LIN {X 0,Y 467.549,Z 320.867,A -85,B 0,C 180,E1 -7525.167,E2 -7525.167} C_VEL
LIN {X 0,Y 467.574,Z 320.867,A -85,B 0,C 180,E1 -7528.26,E2 -7528.26} C_VEL
LIN {X 0,Y 467.538,Z 320.867,A -85,B 0,C 180,E1 -7531.248,E2 -7531.248} C_VEL
LIN {X 0,Y 467.578,Z 320.87,A -85,B 0,C 180,E1 -7534.401,E2 -7534.401} C_VEL
LIN {X 0,Y 467.552,Z 320.866,A -85,B 0,C 180,E1 -7536.995,E2 -7536.995} C_VEL
LIN {X 0,Y 467.613,Z 320.859,A -85,B 0,C 180,E1 -7539.777,E2 -7539.777} C_VEL
LIN {X 0,Y 467.566,Z 320.868,A -85,B 0,C 180,E1 -7542.505,E2 -7542.505} C_VEL
LIN {X 0,Y 467.593,Z 320.86,A -85,B 0,C 180,E1 -7545.196,E2 -7545.196} C_VEL
LIN {X 0,Y 467.658,Z 320.855,A -85,B 0,C 180,E1 -7547.855,E2 -7547.855} C_VEL
LIN {X 0,Y 467.669,Z 320.851,A -85,B 0,C 180,E1 -7551.357,E2 -7551.357} C_VEL
LIN {X 0,Y 467.719,Z 320.851,A -85,B 0,C 180,E1 -7553.963,E2 -7553.963} C_VEL
LIN {X 0,Y 467.852,Z 320.829,A -85,B 0,C 180,E1 -7557.417,E2 -7557.417} C_VEL
LIN {X 0,Y 467.881,Z 320.832,A -85,B 0,C 180,E1 -7560,E2 -7560} C_VEL
LIN {X 0,Y 467.85,Z 320.829,A -85,B 0,C 180,E1 -7562.583,E2 -7562.583} C_VEL
LIN {X 0,Y 467.723,Z 320.85,A -85,B 0,C 180,E1 -7566.038,E2 -7566.038} C_VEL
LIN {X 0,Y 467.683,Z 320.849,A -85,B 0,C 180,E1 -7568.643,E2 -7568.643} C_VEL
LIN {X 0,Y 467.658,Z 320.853,A -85,B 0,C 180,E1 -7572.358,E2 -7572.358} C_VEL
LIN {X 0,Y 467.653,Z 320.858,A -85,B 0,C 180,E1 -7575.885,E2 -7575.885} C_VEL
LIN {X 0,Y 467.627,Z 320.859,A -85,B 0,C 180,E1 -7579.308,E2 -7579.308} C_VEL
LIN {X 0,Y 467.538,Z 320.869,A -85,B 0,C 180,E1 -7582.074,E2 -7582.074} C_VEL
LIN {X 0,Y 467.589,Z 320.861,A -85,B 0,C 180,E1 -7584.888,E2 -7584.888} C_VEL
LIN {X 0,Y 467.624,Z 320.861,A -85,B 0,C 180,E1 -7587.769,E2 -7587.769} C_VEL
LIN {X 0,Y 467.572,Z 320.865,A -85,B 0,C 180,E1 -7591.045,E2 -7591.045} C_VEL
LIN {X 0,Y 467.591,Z 320.86,A -85,B 0,C 180,E1 -7594.242,E2 -7594.242} C_VEL
LIN {X 0,Y 467.546,Z 320.871,A -85,B 0,C 180,E1 -7597.185,E2 -7597.185} C_VEL
LIN {X 0,Y 467.581,Z 320.861,A -85,B 0,C 180,E1 -7600.264,E2 -7600.264} C_VEL
LIN {X 0,Y 467.591,Z 320.861,A -85,B 0,C 180,E1 -7602.567,E2 -7602.567} C_VEL
LIN {X 0,Y 467.574,Z 320.868,A -85,B 0,C 180,E1 -7605.053,E2 -7605.053} C_VEL
LIN {X 0,Y 467.593,Z 320.865,A -85,B 0,C 180,E1 -7607.44,E2 -7607.44} C_VEL
LIN {X 0,Y 467.586,Z 320.865,A -85,B 0,C 180,E1 -7610.855,E2 -7610.855} C_VEL
LIN {X 0,Y 467.564,Z 320.864,A -85,B 0,C 180,E1 -7614.261,E2 -7614.261} C_VEL
LIN {X 0,Y 467.586,Z 320.867,A -85,B 0,C 180,E1 -7617.321,E2 -7617.321} C_VEL
LIN {X 0,Y 467.573,Z 320.872,A -85,B 0,C 180,E1 -7620.667,E2 -7620.667} C_VEL
LIN {X 0,Y 467.642,Z 320.956,A -85,B 0,C 180,E1 -7621.714,E2 -7621.714} C_VEL
LIN {X 0,Y 470.915,Z 336.083,A -85,B 0,C 180,E1 -7624.354,E2 -7624.354} C_VEL
LIN {X 0,Y 470.576,Z 345.926,A -85,B 0,C 180,E1 -7625.915,E2 -7625.915} C_VEL
LIN {X 0,Y 469.657,Z 365.378,A -85,B 0,C 180,E1 -7628.952,E2 -7628.952} C_VEL
LIN {X 0,Y 469.514,Z 368.376,A -85,B 0,C 180,E1 -7629.416,E2 -7629.416} C_VEL
LIN {X 0,Y 473.317,Z 391.092,A -85,B 0,C 180,E1 -7629.937,E2 -7629.937} C_VEL
LIN {X 0,Y 472.11,Z 506.208,A -85,B 0,C 180,E1 -7631.726,E2 -7631.726} C_VEL
LIN {X 0,Y 471.675,Z 521.021,A -85,B 0,C 180,E1 -7632.13,E2 -7632.13} C_VEL
LIN {X 0,Y 471.143,Z 534.853,A -85,B 0,C 180,E1 -7632.686,E2 -7632.686} C_VEL
LIN {X 0,Y 470.514,Z 548.55,A -85,B 0,C 180,E1 -7633.425,E2 -7633.425} C_VEL
LIN {X 0,Y 469.856,Z 560.834,A -85,B 0,C 180,E1 -7634.269,E2 -7634.269} C_VEL
LIN {X 0,Y 469.176,Z 572.39,A -85,B 0,C 180,E1 -7635.246,E2 -7635.246} C_VEL
LIN {X 0,Y 468.566,Z 582.999,A -85,B 0,C 180,E1 -7636.335,E2 -7636.335} C_VEL
LIN {X 0,Y 468.11,Z 592.848,A -85,B 0,C 180,E1 -7637.552,E2 -7637.552} C_VEL
LIN {X 0,Y 467.575,Z 602.232,A -85,B 0,C 180,E1 -7638.951,E2 -7638.951} C_VEL
LIN {X 0,Y 467.175,Z 610.555,A -85,B 0,C 180,E1 -7640.474,E2 -7640.474} C_VEL
LIN {X 0,Y 466.931,Z 616.367,A -85,B 0,C 180,E1 -7641.778,E2 -7641.778} C_VEL
LIN {X 0,Y 466.801,Z 621.141,A -85,B 0,C 180,E1 -7643.081,E2 -7643.081} C_VEL
LIN {X 0,Y 466.729,Z 626.083,A -85,B 0,C 180,E1 -7644.816,E2 -7644.816} C_VEL
LIN {X 0,Y 466.681,Z 629.517,A -85,B 0,C 180,E1 -7646.546,E2 -7646.546} C_VEL
LIN {X 0,Y 466.629,Z 631.547,A -85,B 0,C 180,E1 -7648.273,E2 -7648.273} C_VEL
LIN {X 0,Y 466.597,Z 632.219,A -85,B 0,C 180,E1 -7649.999,E2 -7649.999} C_VEL
LIN {X 0,Y 466.629,Z 631.545,A -85,B 0,C 180,E1 -7651.725,E2 -7651.725} C_VEL
LIN {X 0,Y 466.681,Z 629.513,A -85,B 0,C 180,E1 -7653.453,E2 -7653.453} C_VEL
LIN {X 0,Y 466.73,Z 626.075,A -85,B 0,C 180,E1 -7655.183,E2 -7655.183} C_VEL
LIN {X 0,Y 466.821,Z 621.129,A -85,B 0,C 180,E1 -7656.917,E2 -7656.917} C_VEL
LIN {X 0,Y 466.997,Z 614.534,A -85,B 0,C 180,E1 -7658.655,E2 -7658.655} C_VEL
LIN {X 0,Y 467.29,Z 607.208,A -85,B 0,C 180,E1 -7660.178,E2 -7660.178} C_VEL
LIN {X 0,Y 467.782,Z 598.156,A -85,B 0,C 180,E1 -7661.701,E2 -7661.701} C_VEL
LIN {X 0,Y 468.297,Z 588.667,A -85,B 0,C 180,E1 -7663.009,E2 -7663.009} C_VEL
LIN {X 0,Y 468.85,Z 578.175,A -85,B 0,C 180,E1 -7664.208,E2 -7664.208} C_VEL
LIN {X 0,Y 469.579,Z 566.617,A -85,B 0,C 180,E1 -7665.294,E2 -7665.294} C_VEL
LIN {X 0,Y 470.318,Z 553.814,A -85,B 0,C 180,E1 -7666.27,E2 -7666.27} C_VEL
LIN {X 0,Y 470.942,Z 541.697,A -85,B 0,C 180,E1 -7667.009,E2 -7667.009} C_VEL
LIN {X 0,Y 471.5,Z 527.504,A -85,B 0,C 180,E1 -7667.679,E2 -7667.679} C_VEL
LIN {X 0,Y 472.075,Z 513.044,A -85,B 0,C 180,E1 -7668.161,E2 -7668.161} C_VEL
LIN {X 0,Y 472.405,Z 498.853,A -85,B 0,C 180,E1 -7668.457,E2 -7668.457} C_VEL
LIN {X 0,Y 473.422,Z 390.059,A -85,B 0,C 180,E1 -7670.149,E2 -7670.149} C_VEL
LIN {X 0,Y 469.586,Z 368.039,A -85,B 0,C 180,E1 -7670.692,E2 -7670.692} C_VEL
LIN {X 0,Y 470.566,Z 349.91,A -85,B 0,C 180,E1 -7673.547,E2 -7673.547} C_VEL
LIN {X 0,Y 471.099,Z 336.963,A -85,B 0,C 180,E1 -7675.634,E2 -7675.634} C_VEL
LIN {X 0,Y 468.366,Z 324.027,A -85,B 0,C 180,E1 -7677.962,E2 -7677.962} C_VEL
LIN {X 0,Y 467.606,Z 320.864,A -85,B 0,C 180,E1 -7678.562,E2 -7678.562} C_VEL
LIN {X 0,Y 467.581,Z 320.864,A -85,B 0,C 180,E1 -7681.739,E2 -7681.739} C_VEL
LIN {X 0,Y 467.566,Z 320.871,A -85,B 0,C 180,E1 -7684.831,E2 -7684.831} C_VEL
LIN {X 0,Y 467.566,Z 320.866,A -85,B 0,C 180,E1 -7688.043,E2 -7688.043} C_VEL
LIN {X 0,Y 467.59,Z 320.865,A -85,B 0,C 180,E1 -7690.262,E2 -7690.262} C_VEL
LIN {X 0,Y 467.582,Z 320.862,A -85,B 0,C 180,E1 -7692.566,E2 -7692.566} C_VEL
LIN {X 0,Y 467.566,Z 320.862,A -85,B 0,C 180,E1 -7695.052,E2 -7695.052} C_VEL
LIN {X 0,Y 467.584,Z 320.863,A -85,B 0,C 180,E1 -7697.439,E2 -7697.439} C_VEL
LIN {X 0,Y 467.577,Z 320.861,A -85,B 0,C 180,E1 -7700.854,E2 -7700.854} C_VEL
LIN {X 0,Y 467.557,Z 320.869,A -85,B 0,C 180,E1 -7704.26,E2 -7704.26} C_VEL
LIN {X 0,Y 467.575,Z 320.861,A -85,B 0,C 180,E1 -7707.32,E2 -7707.32} C_VEL
LIN {X 0,Y 467.572,Z 320.867,A -85,B 0,C 180,E1 -7710.665,E2 -7710.665} C_VEL
LIN {X 0,Y 467.619,Z 320.855,A -85,B 0,C 180,E1 -7713.2,E2 -7713.2} C_VEL
LIN {X 0,Y 467.584,Z 320.863,A -85,B 0,C 180,E1 -7716.468,E2 -7716.468} C_VEL
LIN {X 0,Y 467.615,Z 320.862,A -85,B 0,C 180,E1 -7719.777,E2 -7719.777} C_VEL
LIN {X 0,Y 467.601,Z 320.863,A -85,B 0,C 180,E1 -7722.506,E2 -7722.506} C_VEL
LIN {X 0,Y 467.597,Z 320.856,A -85,B 0,C 180,E1 -7725.196,E2 -7725.196} C_VEL
LIN {X 0,Y 467.647,Z 320.86,A -85,B 0,C 180,E1 -7727.854,E2 -7727.854} C_VEL
LIN {X 0,Y 467.67,Z 320.853,A -85,B 0,C 180,E1 -7731.357,E2 -7731.357} C_VEL
LIN {X 0,Y 467.723,Z 320.849,A -85,B 0,C 180,E1 -7733.962,E2 -7733.962} C_VEL
LIN {X 0,Y 467.811,Z 320.834,A -85,B 0,C 180,E1 -7737.417,E2 -7737.417} C_VEL
LIN {X 0,Y 467.839,Z 320.832,A -85,B 0,C 180,E1 -7740,E2 -7740} C_VEL
LIN {X 0,Y 467.837,Z 320.83,A -85,B 0,C 180,E1 -7742.583,E2 -7742.583} C_VEL
LIN {X 0,Y 467.683,Z 320.852,A -85,B 0,C 180,E1 -7746.038,E2 -7746.038} C_VEL
LIN {X 0,Y 467.624,Z 320.855,A -85,B 0,C 180,E1 -7748.644,E2 -7748.644} C_VEL
LIN {X 0,Y 467.645,Z 320.852,A -85,B 0,C 180,E1 -7752.145,E2 -7752.145} C_VEL
LIN {X 0,Y 467.612,Z 320.858,A -85,B 0,C 180,E1 -7755.873,E2 -7755.873} C_VEL
LIN {X 0,Y 467.608,Z 320.863,A -85,B 0,C 180,E1 -7759.308,E2 -7759.308} C_VEL
LIN {X 0,Y 467.52,Z 320.868,A -85,B 0,C 180,E1 -7762.074,E2 -7762.074} C_VEL
LIN {X 0,Y 467.558,Z 320.87,A -85,B 0,C 180,E1 -7764.89,E2 -7764.89} C_VEL
LIN {X 0,Y 467.552,Z 320.863,A -85,B 0,C 180,E1 -7767.773,E2 -7767.773} C_VEL
LIN {X 0,Y 467.555,Z 320.876,A -85,B 0,C 180,E1 -7771.044,E2 -7771.044} C_VEL
LIN {X 0,Y 467.567,Z 320.867,A -85,B 0,C 180,E1 -7774.24,E2 -7774.24} C_VEL
LIN {X 0,Y 467.538,Z 320.872,A -85,B 0,C 180,E1 -7777.187,E2 -7777.187} C_VEL
LIN {X 0,Y 467.566,Z 320.865,A -85,B 0,C 180,E1 -7780.265,E2 -7780.265} C_VEL
LIN {X 0,Y 467.578,Z 320.865,A -85,B 0,C 180,E1 -7782.567,E2 -7782.567} C_VEL
LIN {X 0,Y 467.557,Z 320.871,A -85,B 0,C 180,E1 -7785.053,E2 -7785.053} C_VEL
LIN {X 0,Y 467.623,Z 321.03,A -85,B 0,C 180,E1 -7788.184,E2 -7788.184} C_VEL
LIN {X 0,Y 469.868,Z 332.052,A -85,B 0,C 180,E1 -7790.531,E2 -7790.531} C_VEL
LIN {X 0,Y 469.882,Z 336.532,A -85,B 0,C 180,E1 -7791.386,E2 -7791.386} C_VEL
LIN {X 0,Y 473.693,Z 353.213,A -85,B 0,C 180,E1 -7791.844,E2 -7791.844} C_VEL
LIN {X 0,Y 472.479,Z 472.361,A -85,B 0,C 180,E1 -7793.721,E2 -7793.721} C_VEL
LIN {X 0,Y 472.092,Z 486.72,A -85,B 0,C 180,E1 -7794.115,E2 -7794.115} C_VEL
LIN {X 0,Y 471.664,Z 500.331,A -85,B 0,C 180,E1 -7794.666,E2 -7794.666} C_VEL
LIN {X 0,Y 471.228,Z 510.399,A -85,B 0,C 180,E1 -7795.189,E2 -7795.189} C_VEL
LIN {X 0,Y 470.402,Z 515.734,A -85,B 0,C 180,E1 -7795.48,E2 -7795.48} C_VEL
LIN {X 0,Y 467.231,Z 524.272,A -85,B 0,C 180,E1 -7795.959,E2 -7795.959} C_VEL
LIN {X 0,Y 463.936,Z 532.468,A -85,B 0,C 180,E1 -7796.514,E2 -7796.514} C_VEL
LIN {X 0,Y 462.926,Z 537.249,A -85,B 0,C 180,E1 -7796.923,E2 -7796.923} C_VEL
LIN {X 0,Y 462.295,Z 547.807,A -85,B 0,C 180,E1 -7798.021,E2 -7798.021} C_VEL
LIN {X 0,Y 461.603,Z 558.262,A -85,B 0,C 180,E1 -7799.334,E2 -7799.334} C_VEL
LIN {X 0,Y 460.96,Z 567.82,A -85,B 0,C 180,E1 -7800.799,E2 -7800.799} C_VEL
LIN {X 0,Y 460.489,Z 575.654,A -85,B 0,C 180,E1 -7802.275,E2 -7802.275} C_VEL
LIN {X 0,Y 460.121,Z 581.847,A -85,B 0,C 180,E1 -7803.709,E2 -7803.709} C_VEL
LIN {X 0,Y 459.901,Z 586.868,A -85,B 0,C 180,E1 -7805.151,E2 -7805.151} C_VEL
LIN {X 0,Y 459.725,Z 590.787,A -85,B 0,C 180,E1 -7806.581,E2 -7806.581} C_VEL
LIN {X 0,Y 459.556,Z 594.49,A -85,B 0,C 180,E1 -7808.468,E2 -7808.468} C_VEL
LIN {X 0,Y 459.491,Z 596.599,A -85,B 0,C 180,E1 -7810.338,E2 -7810.338} C_VEL
LIN {X 0,Y 459.481,Z 597.172,A -85,B 0,C 180,E1 -7812.188,E2 -7812.188} C_VEL
LIN {X 0,Y 459.454,Z 596.31,A -85,B 0,C 180,E1 -7814.019,E2 -7814.019} C_VEL
LIN {X 0,Y 459.544,Z 594.028,A -85,B 0,C 180,E1 -7815.837,E2 -7815.837} C_VEL
LIN {X 0,Y 459.75,Z 590.297,A -85,B 0,C 180,E1 -7817.643,E2 -7817.643} C_VEL
LIN {X 0,Y 459.96,Z 585.044,A -85,B 0,C 180,E1 -7819.436,E2 -7819.436} C_VEL
LIN {X 0,Y 460.2,Z 579.947,A -85,B 0,C 180,E1 -7820.774,E2 -7820.774} C_VEL
LIN {X 0,Y 460.54,Z 573.802,A -85,B 0,C 180,E1 -7822.107,E2 -7822.107} C_VEL
LIN {X 0,Y 461.059,Z 565.093,A -85,B 0,C 180,E1 -7823.656,E2 -7823.656} C_VEL
LIN {X 0,Y 461.579,Z 556.016,A -85,B 0,C 180,E1 -7824.978,E2 -7824.978} C_VEL
LIN {X 0,Y 462.27,Z 545.023,A -85,B 0,C 180,E1 -7826.296,E2 -7826.296} C_VEL
LIN {X 0,Y 462.964,Z 533.821,A -85,B 0,C 180,E1 -7827.391,E2 -7827.391} C_VEL
LIN {X 0,Y 463.685,Z 521.54,A -85,B 0,C 180,E1 -7828.367,E2 -7828.367} C_VEL
LIN {X 0,Y 464.295,Z 509.57,A -85,B 0,C 180,E1 -7829.133,E2 -7829.133} C_VEL
LIN {X 0,Y 464.848,Z 496.574,A -85,B 0,C 180,E1 -7829.784,E2 -7829.784} C_VEL
LIN {X 0,Y 465.285,Z 482.579,A -85,B 0,C 180,E1 -7830.298,E2 -7830.298} C_VEL
LIN {X 0,Y 465.603,Z 467.783,A -85,B 0,C 180,E1 -7830.649,E2 -7830.649} C_VEL
LIN {X 0,Y 466.765,Z 354.137,A -85,B 0,C 180,E1 -7832.433,E2 -7832.433} C_VEL
LIN {X 0,Y 462.828,Z 336.193,A -85,B 0,C 180,E1 -7832.917,E2 -7832.917} C_VEL
LIN {X 0,Y 462.659,Z 332.235,A -85,B 0,C 180,E1 -7833.702,E2 -7833.702} C_VEL
LIN {X 0,Y 460.676,Z 321.729,A -85,B 0,C 180,E1 -7835.911,E2 -7835.911} C_VEL
LIN {X 0,Y 460.615,Z 321.735,A -85,B 0,C 180,E1 -7838.777,E2 -7838.777} C_VEL
LIN {X 0,Y 460.595,Z 321.732,A -85,B 0,C 180,E1 -7842.436,E2 -7842.436} C_VEL
LIN {X 0,Y 460.599,Z 321.732,A -85,B 0,C 180,E1 -7845.998,E2 -7845.998} C_VEL
LIN {X 0,Y 460.566,Z 321.738,A -85,B 0,C 180,E1 -7849.616,E2 -7849.616} C_VEL
LIN {X 0,Y 460.505,Z 321.744,A -85,B 0,C 180,E1 -7852.43,E2 -7852.43} C_VEL
LIN {X 0,Y 460.531,Z 321.74,A -85,B 0,C 180,E1 -7855.793,E2 -7855.793} C_VEL
LIN {X 0,Y 460.513,Z 321.747,A -85,B 0,C 180,E1 -7859.233,E2 -7859.233} C_VEL
LIN {X 0,Y 460.497,Z 321.745,A -85,B 0,C 180,E1 -7862.288,E2 -7862.288} C_VEL
LIN {X 0,Y 460.497,Z 321.746,A -85,B 0,C 180,E1 -7865.447,E2 -7865.447} C_VEL
LIN {X 0,Y 460.488,Z 321.753,A -85,B 0,C 180,E1 -7868.89,E2 -7868.89} C_VEL
LIN {X 0,Y 460.5,Z 321.744,A -85,B 0,C 180,E1 -7871.599,E2 -7871.599} C_VEL
LIN {X 0,Y 460.509,Z 321.748,A -85,B 0,C 180,E1 -7874.59,E2 -7874.59} C_VEL
LIN {X 0,Y 460.471,Z 321.747,A -85,B 0,C 180,E1 -7877.813,E2 -7877.813} C_VEL
LIN {X 0,Y 460.475,Z 321.749,A -85,B 0,C 180,E1 -7880.132,E2 -7880.132} C_VEL
LIN {X 0,Y 460.457,Z 321.749,A -85,B 0,C 180,E1 -7883.469,E2 -7883.469} C_VEL
LIN {X 0,Y 460.516,Z 321.748,A -85,B 0,C 180,E1 -7886.675,E2 -7886.675} C_VEL
LIN {X 0,Y 460.496,Z 321.745,A -85,B 0,C 180,E1 -7889.759,E2 -7889.759} C_VEL
LIN {X 0,Y 460.49,Z 321.749,A -85,B 0,C 180,E1 -7892.751,E2 -7892.751} C_VEL
LIN {X 0,Y 460.516,Z 321.742,A -85,B 0,C 180,E1 -7895.667,E2 -7895.667} C_VEL
LIN {X 0,Y 460.52,Z 321.746,A -85,B 0,C 180,E1 -7898.58,E2 -7898.58} C_VEL
LIN {X 0,Y 460.584,Z 321.733,A -85,B 0,C 180,E1 -7901.311,E2 -7901.311} C_VEL
LIN {X 0,Y 460.55,Z 321.738,A -85,B 0,C 180,E1 -7904.965,E2 -7904.965} C_VEL
LIN {X 0,Y 460.611,Z 321.733,A -85,B 0,C 180,E1 -7908.56,E2 -7908.56} C_VEL
LIN {X 0,Y 460.62,Z 321.729,A -85,B 0,C 180,E1 -7911.224,E2 -7911.224} C_VEL
LIN {X 0,Y 460.683,Z 321.726,A -85,B 0,C 180,E1 -7913.87,E2 -7913.87} C_VEL
LIN {X 0,Y 460.793,Z 321.708,A -85,B 0,C 180,E1 -7917.378,E2 -7917.378} C_VEL
LIN {X 0,Y 460.85,Z 321.708,A -85,B 0,C 180,E1 -7920,E2 -7920} C_VEL
LIN {X 0,Y 460.79,Z 321.708,A -85,B 0,C 180,E1 -7922.623,E2 -7922.623} C_VEL
LIN {X 0,Y 460.687,Z 321.725,A -85,B 0,C 180,E1 -7926.13,E2 -7926.13} C_VEL
LIN {X 0,Y 460.63,Z 321.727,A -85,B 0,C 180,E1 -7928.776,E2 -7928.776} C_VEL
LIN {X 0,Y 460.6,Z 321.732,A -85,B 0,C 180,E1 -7932.435,E2 -7932.435} C_VEL
LIN {X 0,Y 460.604,Z 321.735,A -85,B 0,C 180,E1 -7935.998,E2 -7935.998} C_VEL
LIN {X 0,Y 460.575,Z 321.735,A -85,B 0,C 180,E1 -7938.902,E2 -7938.902} C_VEL
LIN {X 0,Y 460.52,Z 321.747,A -85,B 0,C 180,E1 -7941.486,E2 -7941.486} C_VEL
LIN {X 0,Y 460.535,Z 321.74,A -85,B 0,C 180,E1 -7944.333,E2 -7944.333} C_VEL
LIN {X 0,Y 460.575,Z 321.738,A -85,B 0,C 180,E1 -7947.244,E2 -7947.244} C_VEL
LIN {X 0,Y 460.514,Z 321.742,A -85,B 0,C 180,E1 -7950.24,E2 -7950.24} C_VEL
LIN {X 0,Y 460.533,Z 321.746,A -85,B 0,C 180,E1 -7953.325,E2 -7953.325} C_VEL
LIN {X 0,Y 460.476,Z 321.747,A -85,B 0,C 180,E1 -7956.53,E2 -7956.53} C_VEL
LIN {X 0,Y 460.536,Z 321.741,A -85,B 0,C 180,E1 -7959.862,E2 -7959.862} C_VEL
LIN {X 0,Y 460.521,Z 321.744,A -85,B 0,C 180,E1 -7962.901,E2 -7962.901} C_VEL
LIN {X 0,Y 460.515,Z 321.743,A -85,B 0,C 180,E1 -7965.83,E2 -7965.83} C_VEL
LIN {X 0,Y 460.535,Z 321.745,A -85,B 0,C 180,E1 -7968.989,E2 -7968.989} C_VEL
LIN {X 0,Y 460.531,Z 321.746,A -85,B 0,C 180,E1 -7971.267,E2 -7971.267} C_VEL
LIN {X 0,Y 460.515,Z 321.744,A -85,B 0,C 180,E1 -7974.554,E2 -7974.554} C_VEL
LIN {X 0,Y 460.535,Z 321.745,A -85,B 0,C 180,E1 -7977.715,E2 -7977.715} C_VEL
LIN {X 0,Y 460.556,Z 321.747,A -85,B 0,C 180,E1 -7981.269,E2 -7981.269} C_VEL
LIN {X 0,Y 460.573,Z 321.799,A -85,B 0,C 180,E1 -7981.457,E2 -7981.457} C_VEL
LIN {X 0,Y 463.649,Z 335.663,A -85,B 0,C 180,E1 -7983.922,E2 -7983.922} C_VEL
LIN {X 0,Y 464.112,Z 338.642,A -85,B 0,C 180,E1 -7984.432,E2 -7984.432} C_VEL
LIN {X 0,Y 463.063,Z 359.71,A -85,B 0,C 180,E1 -7987.791,E2 -7987.791} C_VEL
LIN {X 0,Y 462.599,Z 368.072,A -85,B 0,C 180,E1 -7989.107,E2 -7989.107} C_VEL
LIN {X 0,Y 466.604,Z 392.316,A -85,B 0,C 180,E1 -7989.677,E2 -7989.677} C_VEL
LIN {X 0,Y 465.34,Z 506.543,A -85,B 0,C 180,E1 -7991.479,E2 -7991.479} C_VEL
LIN {X 0,Y 464.873,Z 521.131,A -85,B 0,C 180,E1 -7991.888,E2 -7991.888} C_VEL
LIN {X 0,Y 464.314,Z 534.485,A -85,B 0,C 180,E1 -7992.432,E2 -7992.432} C_VEL
LIN {X 0,Y 463.677,Z 548.174,A -85,B 0,C 180,E1 -7993.181,E2 -7993.181} C_VEL
LIN {X 0,Y 462.99,Z 560.386,A -85,B 0,C 180,E1 -7994.03,E2 -7994.03} C_VEL
LIN {X 0,Y 462.253,Z 571.973,A -85,B 0,C 180,E1 -7995.02,E2 -7995.02} C_VEL
LIN {X 0,Y 461.599,Z 582.607,A -85,B 0,C 180,E1 -7996.125,E2 -7996.125} C_VEL
LIN {X 0,Y 461.083,Z 593.193,A -85,B 0,C 180,E1 -7997.457,E2 -7997.457} C_VEL
LIN {X 0,Y 460.564,Z 601.887,A -85,B 0,C 180,E1 -7998.78,E2 -7998.78} C_VEL
LIN {X 0,Y 460.102,Z 610.237,A -85,B 0,C 180,E1 -8000.326,E2 -8000.326} C_VEL
LIN {X 0,Y 459.85,Z 616.063,A -85,B 0,C 180,E1 -8001.651,E2 -8001.651} C_VEL
LIN {X 0,Y 459.721,Z 620.849,A -85,B 0,C 180,E1 -8002.974,E2 -8002.974} C_VEL
LIN {X 0,Y 459.638,Z 625.801,A -85,B 0,C 180,E1 -8004.735,E2 -8004.735} C_VEL
LIN {X 0,Y 459.578,Z 629.242,A -85,B 0,C 180,E1 -8006.492,E2 -8006.492} C_VEL
LIN {X 0,Y 459.54,Z 631.276,A -85,B 0,C 180,E1 -8008.246,E2 -8008.246} C_VEL
LIN {X 0,Y 459.528,Z 631.951,A -85,B 0,C 180,E1 -8009.999,E2 -8009.999} C_VEL
LIN {X 0,Y 459.54,Z 631.279,A -85,B 0,C 180,E1 -8011.752,E2 -8011.752} C_VEL
LIN {X 0,Y 459.577,Z 629.25,A -85,B 0,C 180,E1 -8013.506,E2 -8013.506} C_VEL
LIN {X 0,Y 459.64,Z 625.817,A -85,B 0,C 180,E1 -8015.263,E2 -8015.263} C_VEL
LIN {X 0,Y 459.73,Z 620.88,A -85,B 0,C 180,E1 -8017.024,E2 -8017.024} C_VEL
LIN {X 0,Y 459.941,Z 614.3,A -85,B 0,C 180,E1 -8018.788,E2 -8018.788} C_VEL
LIN {X 0,Y 460.265,Z 606.988,A -85,B 0,C 180,E1 -8020.335,E2 -8020.335} C_VEL
LIN {X 0,Y 460.761,Z 597.951,A -85,B 0,C 180,E1 -8021.882,E2 -8021.882} C_VEL
LIN {X 0,Y 461.332,Z 588.477,A -85,B 0,C 180,E1 -8023.209,E2 -8023.209} C_VEL
LIN {X 0,Y 461.911,Z 578.001,A -85,B 0,C 180,E1 -8024.426,E2 -8024.426} C_VEL
LIN {X 0,Y 462.712,Z 566.464,A -85,B 0,C 180,E1 -8025.527,E2 -8025.527} C_VEL
LIN {X 0,Y 463.475,Z 553.702,A -85,B 0,C 180,E1 -8026.517,E2 -8026.517} C_VEL
LIN {X 0,Y 464.206,Z 541.17,A -85,B 0,C 180,E1 -8027.291,E2 -8027.291} C_VEL
LIN {X 0,Y 464.738,Z 527.569,A -85,B 0,C 180,E1 -8027.945,E2 -8027.945} C_VEL
LIN {X 0,Y 465.342,Z 513.286,A -85,B 0,C 180,E1 -8028.433,E2 -8028.433} C_VEL
LIN {X 0,Y 465.708,Z 499.57,A -85,B 0,C 180,E1 -8028.732,E2 -8028.732} C_VEL
LIN {X 0,Y 466.861,Z 391.399,A -85,B 0,C 180,E1 -8030.439,E2 -8030.439} C_VEL
LIN {X 0,Y 462.727,Z 367.655,A -85,B 0,C 180,E1 -8031.052,E2 -8031.052} C_VEL
LIN {X 0,Y 463.67,Z 351.255,A -85,B 0,C 180,E1 -8033.681,E2 -8033.681} C_VEL
LIN {X 0,Y 464.338,Z 339.764,A -85,B 0,C 180,E1 -8035.553,E2 -8035.553} C_VEL
LIN {X 0,Y 462.491,Z 329.885,A -85,B 0,C 180,E1 -8037.337,E2 -8037.337} C_VEL
LIN {X 0,Y 460.542,Z 321.744,A -85,B 0,C 180,E1 -8038.917,E2 -8038.917} C_VEL
LIN {X 0,Y 460.529,Z 321.743,A -85,B 0,C 180,E1 -8042.283,E2 -8042.283} C_VEL
LIN {X 0,Y 460.511,Z 321.744,A -85,B 0,C 180,E1 -8045.444,E2 -8045.444} C_VEL
LIN {X 0,Y 460.56,Z 321.739,A -85,B 0,C 180,E1 -8048.9,E2 -8048.9} C_VEL
LIN {X 0,Y 460.52,Z 321.74,A -85,B 0,C 180,E1 -8052.18,E2 -8052.18} C_VEL
LIN {X 0,Y 460.515,Z 321.737,A -85,B 0,C 180,E1 -8055.411,E2 -8055.411} C_VEL
LIN {X 0,Y 460.53,Z 321.747,A -85,B 0,C 180,E1 -8058.396,E2 -8058.396} C_VEL
LIN {X 0,Y 460.521,Z 321.74,A -85,B 0,C 180,E1 -8061.266,E2 -8061.266} C_VEL
LIN {X 0,Y 460.507,Z 321.748,A -85,B 0,C 180,E1 -8064.554,E2 -8064.554} C_VEL
LIN {X 0,Y 460.526,Z 321.74,A -85,B 0,C 180,E1 -8067.715,E2 -8067.715} C_VEL
LIN {X 0,Y 460.541,Z 321.742,A -85,B 0,C 180,E1 -8070.769,E2 -8070.769} C_VEL
LIN {X 0,Y 460.557,Z 321.737,A -85,B 0,C 180,E1 -8073.734,E2 -8073.734} C_VEL
LIN {X 0,Y 460.538,Z 321.738,A -85,B 0,C 180,E1 -8076.623,E2 -8076.623} C_VEL
LIN {X 0,Y 460.543,Z 321.74,A -85,B 0,C 180,E1 -8079.452,E2 -8079.452} C_VEL
LIN {X 0,Y 460.552,Z 321.744,A -85,B 0,C 180,E1 -8082.23,E2 -8082.23} C_VEL
LIN {X 0,Y 460.56,Z 321.732,A -85,B 0,C 180,E1 -8084.964,E2 -8084.964} C_VEL
LIN {X 0,Y 460.6,Z 321.728,A -85,B 0,C 180,E1 -8088.559,E2 -8088.559} C_VEL
LIN {X 0,Y 460.686,Z 321.722,A -85,B 0,C 180,E1 -8092.108,E2 -8092.108} C_VEL
LIN {X 0,Y 460.682,Z 321.722,A -85,B 0,C 180,E1 -8094.748,E2 -8094.748} C_VEL
LIN {X 0,Y 460.755,Z 321.712,A -85,B 0,C 180,E1 -8097.377,E2 -8097.377} C_VEL
LIN {X 0,Y 460.808,Z 321.708,A -85,B 0,C 180,E1 -8100,E2 -8100} C_VEL
LIN {X 0,Y 460.777,Z 321.71,A -85,B 0,C 180,E1 -8102.622,E2 -8102.622} C_VEL
LIN {X 0,Y 460.649,Z 321.728,A -85,B 0,C 180,E1 -8106.13,E2 -8106.13} C_VEL
LIN {X 0,Y 460.579,Z 321.733,A -85,B 0,C 180,E1 -8108.777,E2 -8108.777} C_VEL
LIN {X 0,Y 460.599,Z 321.729,A -85,B 0,C 180,E1 -8112.334,E2 -8112.334} C_VEL
LIN {X 0,Y 460.569,Z 321.735,A -85,B 0,C 180,E1 -8115.988,E2 -8115.988} C_VEL
LIN {X 0,Y 460.554,Z 321.742,A -85,B 0,C 180,E1 -8119.616,E2 -8119.616} C_VEL
LIN {X 0,Y 460.496,Z 321.743,A -85,B 0,C 180,E1 -8122.429,E2 -8122.429} C_VEL
LIN {X 0,Y 460.537,Z 321.743,A -85,B 0,C 180,E1 -8125.797,E2 -8125.797} C_VEL
LIN {X 0,Y 460.505,Z 321.739,A -85,B 0,C 180,E1 -8128.236,E2 -8128.236} C_VEL
LIN {X 0,Y 460.51,Z 321.75,A -85,B 0,C 180,E1 -8131.283,E2 -8131.283} C_VEL
LIN {X 0,Y 460.513,Z 321.747,A -85,B 0,C 180,E1 -8134.504,E2 -8134.504} C_VEL
LIN {X 0,Y 460.492,Z 321.749,A -85,B 0,C 180,E1 -8137.624,E2 -8137.624} C_VEL
LIN {X 0,Y 460.53,Z 321.742,A -85,B 0,C 180,E1 -8140.269,E2 -8140.269} C_VEL
LIN {X 0,Y 460.488,Z 321.749,A -85,B 0,C 180,E1 -8143.376,E2 -8143.376} C_VEL
LIN {X 0,Y 460.491,Z 321.753,A -85,B 0,C 180,E1 -8146.625,E2 -8146.625} C_VEL
LIN {X 0,Y 460.545,Z 321.794,A -85,B 0,C 180,E1 -8147.865,E2 -8147.865} C_VEL
LIN {X 0,Y 462.961,Z 333.439,A -85,B 0,C 180,E1 -8150.39,E2 -8150.39} C_VEL
LIN {X 0,Y 463.049,Z 336.579,A -85,B 0,C 180,E1 -8151.025,E2 -8151.025} C_VEL
LIN {X 0,Y 467.147,Z 354.428,A -85,B 0,C 180,E1 -8151.544,E2 -8151.544} C_VEL
LIN {X 0,Y 465.788,Z 472.967,A -85,B 0,C 180,E1 -8153.437,E2 -8153.437} C_VEL
LIN {X 0,Y 465.387,Z 487.652,A -85,B 0,C 180,E1 -8153.854,E2 -8153.854} C_VEL
LIN {X 0,Y 464.931,Z 500.81,A -85,B 0,C 180,E1 -8154.399,E2 -8154.399} C_VEL
LIN {X 0,Y 464.297,Z 514.458,A -85,B 0,C 180,E1 -8155.152,E2 -8155.152} C_VEL
LIN {X 0,Y 463.543,Z 527.641,A -85,B 0,C 180,E1 -8156.087,E2 -8156.087} C_VEL
LIN {X 0,Y 462.926,Z 537.249,A -85,B 0,C 180,E1 -8156.923,E2 -8156.923} C_VEL
LIN {X 0,Y 461.939,Z 541.954,A -85,B 0,C 180,E1 -8157.355,E2 -8157.355} C_VEL
LIN {X 0,Y 458.704,Z 549.411,A -85,B 0,C 180,E1 -8158.062,E2 -8158.062} C_VEL
LIN {X 0,Y 455.498,Z 556.423,A -85,B 0,C 180,E1 -8158.84,E2 -8158.84} C_VEL
LIN {X 0,Y 454.567,Z 560.365,A -85,B 0,C 180,E1 -8159.38,E2 -8159.38} C_VEL
LIN {X 0,Y 453.911,Z 569.233,A -85,B 0,C 180,E1 -8160.81,E2 -8160.81} C_VEL
LIN {X 0,Y 453.448,Z 576.759,A -85,B 0,C 180,E1 -8162.293,E2 -8162.293} C_VEL
LIN {X 0,Y 453.053,Z 582.828,A -85,B 0,C 180,E1 -8163.753,E2 -8163.753} C_VEL
LIN {X 0,Y 452.822,Z 587.752,A -85,B 0,C 180,E1 -8165.226,E2 -8165.226} C_VEL
LIN {X 0,Y 452.687,Z 590.73,A -85,B 0,C 180,E1 -8166.344,E2 -8166.344} C_VEL
LIN {X 0,Y 452.471,Z 594.303,A -85,B 0,C 180,E1 -8168.114,E2 -8168.114} C_VEL
LIN {X 0,Y 452.39,Z 596.627,A -85,B 0,C 180,E1 -8170.016,E2 -8170.016} C_VEL
LIN {X 0,Y 452.383,Z 597.451,A -85,B 0,C 180,E1 -8171.899,E2 -8171.899} C_VEL
LIN {X 0,Y 452.358,Z 596.823,A -85,B 0,C 180,E1 -8173.761,E2 -8173.761} C_VEL
LIN {X 0,Y 452.45,Z 595.954,A -85,B 0,C 180,E1 -8174.69,E2 -8174.69} C_VEL
LIN {X 0,Y 452.512,Z 593.159,A -85,B 0,C 180,E1 -8176.529,E2 -8176.529} C_VEL
LIN {X 0,Y 452.76,Z 588.881,A -85,B 0,C 180,E1 -8178.359,E2 -8178.359} C_VEL
LIN {X 0,Y 452.994,Z 583.04,A -85,B 0,C 180,E1 -8180.175,E2 -8180.175} C_VEL
LIN {X 0,Y 453.378,Z 576.457,A -85,B 0,C 180,E1 -8181.757,E2 -8181.757} C_VEL
LIN {X 0,Y 453.834,Z 568.322,A -85,B 0,C 180,E1 -8183.331,E2 -8183.331} C_VEL
LIN {X 0,Y 454.409,Z 559.807,A -85,B 0,C 180,E1 -8184.676,E2 -8184.676} C_VEL
LIN {X 0,Y 455.145,Z 549.492,A -85,B 0,C 180,E1 -8186.016,E2 -8186.016} C_VEL
LIN {X 0,Y 455.757,Z 539.194,A -85,B 0,C 180,E1 -8187.128,E2 -8187.128} C_VEL
LIN {X 0,Y 456.511,Z 527.969,A -85,B 0,C 180,E1 -8188.126,E2 -8188.126} C_VEL
LIN {X 0,Y 457.17,Z 515.886,A -85,B 0,C 180,E1 -8189.003,E2 -8189.003} C_VEL
LIN {X 0,Y 457.85,Z 502.212,A -85,B 0,C 180,E1 -8189.781,E2 -8189.781} C_VEL
LIN {X 0,Y 458.336,Z 488.738,A -85,B 0,C 180,E1 -8190.358,E2 -8190.358} C_VEL
LIN {X 0,Y 458.694,Z 474.979,A -85,B 0,C 180,E1 -8190.769,E2 -8190.769} C_VEL
LIN {X 0,Y 459.035,Z 449.705,A -85,B 0,C 180,E1 -8191.207,E2 -8191.207} C_VEL
LIN {X 0,Y 459.968,Z 354.723,A -85,B 0,C 180,E1 -8192.72,E2 -8192.72} C_VEL
LIN {X 0,Y 455.97,Z 336.545,A -85,B 0,C 180,E1 -8193.204,E2 -8193.204} C_VEL
LIN {X 0,Y 455.539,Z 332.748,A -85,B 0,C 180,E1 -8193.982,E2 -8193.982} C_VEL
LIN {X 0,Y 453.652,Z 322.604,A -85,B 0,C 180,E1 -8196.115,E2 -8196.115} C_VEL
LIN {X 0,Y 453.581,Z 322.612,A -85,B 0,C 180,E1 -8198.914,E2 -8198.914} C_VEL
LIN {X 0,Y 453.562,Z 322.608,A -85,B 0,C 180,E1 -8202.53,E2 -8202.53} C_VEL
LIN {X 0,Y 453.543,Z 322.61,A -85,B 0,C 180,E1 -8206.197,E2 -8206.197} C_VEL
LIN {X 0,Y 453.515,Z 322.62,A -85,B 0,C 180,E1 -8209.04,E2 -8209.04} C_VEL
LIN {X 0,Y 453.474,Z 322.619,A -85,B 0,C 180,E1 -8211.837,E2 -8211.837} C_VEL
LIN {X 0,Y 453.466,Z 322.623,A -85,B 0,C 180,E1 -8214.738,E2 -8214.738} C_VEL
LIN {X 0,Y 453.459,Z 322.621,A -85,B 0,C 180,E1 -8217.943,E2 -8217.943} C_VEL
LIN {X 0,Y 453.451,Z 322.627,A -85,B 0,C 180,E1 -8220.762,E2 -8220.762} C_VEL
LIN {X 0,Y 453.453,Z 322.621,A -85,B 0,C 180,E1 -8223.915,E2 -8223.915} C_VEL
LIN {X 0,Y 453.433,Z 322.628,A -85,B 0,C 180,E1 -8227.192,E2 -8227.192} C_VEL
LIN {X 0,Y 453.469,Z 322.625,A -85,B 0,C 180,E1 -8230.612,E2 -8230.612} C_VEL
LIN {X 0,Y 453.479,Z 322.623,A -85,B 0,C 180,E1 -8234.529,E2 -8234.529} C_VEL
LIN {X 0,Y 453.432,Z 322.625,A -85,B 0,C 180,E1 -8238.072,E2 -8238.072} C_VEL
LIN {X 0,Y 453.423,Z 322.631,A -85,B 0,C 180,E1 -8240.805,E2 -8240.805} C_VEL
LIN {X 0,Y 453.44,Z 322.624,A -85,B 0,C 180,E1 -8243.916,E2 -8243.916} C_VEL
LIN {X 0,Y 453.474,Z 322.62,A -85,B 0,C 180,E1 -8247.151,E2 -8247.151} C_VEL
LIN {X 0,Y 453.455,Z 322.626,A -85,B 0,C 180,E1 -8250.267,E2 -8250.267} C_VEL
LIN {X 0,Y 453.442,Z 322.623,A -85,B 0,C 180,E1 -8253.29,E2 -8253.29} C_VEL
LIN {X 0,Y 453.482,Z 322.624,A -85,B 0,C 180,E1 -8256.238,E2 -8256.238} C_VEL
LIN {X 0,Y 453.475,Z 322.619,A -85,B 0,C 180,E1 -8259.118,E2 -8259.118} C_VEL
LIN {X 0,Y 453.487,Z 322.621,A -85,B 0,C 180,E1 -8261.944,E2 -8261.944} C_VEL
LIN {X 0,Y 453.52,Z 322.615,A -85,B 0,C 180,E1 -8264.726,E2 -8264.726} C_VEL
LIN {X 0,Y 453.561,Z 322.613,A -85,B 0,C 180,E1 -8268.379,E2 -8268.379} C_VEL
LIN {X 0,Y 453.586,Z 322.605,A -85,B 0,C 180,E1 -8271.087,E2 -8271.087} C_VEL
LIN {X 0,Y 453.649,Z 322.601,A -85,B 0,C 180,E1 -8273.775,E2 -8273.775} C_VEL
LIN {X 0,Y 453.737,Z 322.587,A -85,B 0,C 180,E1 -8277.337,E2 -8277.337} C_VEL
LIN {X 0,Y 453.82,Z 322.584,A -85,B 0,C 180,E1 -8280,E2 -8280} C_VEL
LIN {X 0,Y 453.734,Z 322.587,A -85,B 0,C 180,E1 -8282.664,E2 -8282.664} C_VEL
LIN {X 0,Y 453.653,Z 322.6,A -85,B 0,C 180,E1 -8286.226,E2 -8286.226} C_VEL
LIN {X 0,Y 453.594,Z 322.604,A -85,B 0,C 180,E1 -8288.914,E2 -8288.914} C_VEL
LIN {X 0,Y 453.568,Z 322.608,A -85,B 0,C 180,E1 -8292.529,E2 -8292.529} C_VEL
LIN {X 0,Y 453.549,Z 322.612,A -85,B 0,C 180,E1 -8296.196,E2 -8296.196} C_VEL
LIN {X 0,Y 453.524,Z 322.614,A -85,B 0,C 180,E1 -8299.041,E2 -8299.041} C_VEL
LIN {X 0,Y 453.48,Z 322.623,A -85,B 0,C 180,E1 -8301.836,E2 -8301.836} C_VEL
LIN {X 0,Y 453.504,Z 322.615,A -85,B 0,C 180,E1 -8304.735,E2 -8304.735} C_VEL
LIN {X 0,Y 453.536,Z 322.614,A -85,B 0,C 180,E1 -8307.959,E2 -8307.959} C_VEL
LIN {X 0,Y 453.47,Z 322.627,A -85,B 0,C 180,E1 -8311.525,E2 -8311.525} C_VEL
LIN {X 0,Y 453.49,Z 322.618,A -85,B 0,C 180,E1 -8314.777,E2 -8314.777} C_VEL
LIN {X 0,Y 453.467,Z 322.62,A -85,B 0,C 180,E1 -8318.312,E2 -8318.312} C_VEL
LIN {X 0,Y 453.498,Z 322.616,A -85,B 0,C 180,E1 -8320.609,E2 -8320.609} C_VEL
LIN {X 0,Y 453.476,Z 322.618,A -85,B 0,C 180,E1 -8324.22,E2 -8324.22} C_VEL
LIN {X 0,Y 453.468,Z 322.625,A -85,B 0,C 180,E1 -8327.005,E2 -8327.005} C_VEL
LIN {X 0,Y 453.498,Z 322.62,A -85,B 0,C 180,E1 -8329.409,E2 -8329.409} C_VEL
LIN {X 0,Y 453.454,Z 322.621,A -85,B 0,C 180,E1 -8332.227,E2 -8332.227} C_VEL
LIN {X 0,Y 453.492,Z 322.622,A -85,B 0,C 180,E1 -8335.222,E2 -8335.222} C_VEL
LIN {X 0,Y 453.469,Z 322.626,A -85,B 0,C 180,E1 -8338.475,E2 -8338.475} C_VEL
LIN {X 0,Y 453.509,Z 322.641,A -85,B 0,C 180,E1 -8341.193,E2 -8341.193} C_VEL
LIN {X 0,Y 456.665,Z 336.702,A -85,B 0,C 180,E1 -8343.739,E2 -8343.739} C_VEL
LIN {X 0,Y 457.166,Z 341.159,A -85,B 0,C 180,E1 -8344.504,E2 -8344.504} C_VEL
LIN {X 0,Y 456.115,Z 361.079,A -85,B 0,C 180,E1 -8347.721,E2 -8347.721} C_VEL
LIN {X 0,Y 455.696,Z 367.823,A -85,B 0,C 180,E1 -8348.797,E2 -8348.797} C_VEL
LIN {X 0,Y 459.888,Z 393.017,A -85,B 0,C 180,E1 -8349.401,E2 -8349.401} C_VEL
LIN {X 0,Y 458.563,Z 506.621,A -85,B 0,C 180,E1 -8351.225,E2 -8351.225} C_VEL
LIN {X 0,Y 458.073,Z 521.111,A -85,B 0,C 180,E1 -8351.638,E2 -8351.638} C_VEL
LIN {X 0,Y 457.476,Z 534.751,A -85,B 0,C 180,E1 -8352.207,E2 -8352.207} C_VEL
LIN {X 0,Y 456.843,Z 547.767,A -85,B 0,C 180,E1 -8352.93,E2 -8352.93} C_VEL
LIN {X 0,Y 456.086,Z 559.916,A -85,B 0,C 180,E1 -8353.781,E2 -8353.781} C_VEL
LIN {X 0,Y 455.355,Z 571.557,A -85,B 0,C 180,E1 -8354.788,E2 -8354.788} C_VEL
LIN {X 0,Y 454.653,Z 582.216,A -85,B 0,C 180,E1 -8355.908,E2 -8355.908} C_VEL
LIN {X 0,Y 454.078,Z 592.268,A -85,B 0,C 180,E1 -8357.184,E2 -8357.184} C_VEL
LIN {X 0,Y 453.547,Z 601.535,A -85,B 0,C 180,E1 -8358.604,E2 -8358.604} C_VEL
LIN {X 0,Y 453.039,Z 609.905,A -85,B 0,C 180,E1 -8360.174,E2 -8360.174} C_VEL
LIN {X 0,Y 452.789,Z 615.74,A -85,B 0,C 180,E1 -8361.52,E2 -8361.52} C_VEL
LIN {X 0,Y 452.645,Z 620.539,A -85,B 0,C 180,E1 -8362.864,E2 -8362.864} C_VEL
LIN {X 0,Y 452.548,Z 625.502,A -85,B 0,C 180,E1 -8364.653,E2 -8364.653} C_VEL
LIN {X 0,Y 452.476,Z 628.953,A -85,B 0,C 180,E1 -8366.437,E2 -8366.437} C_VEL
LIN {X 0,Y 452.455,Z 630.997,A -85,B 0,C 180,E1 -8368.219,E2 -8368.219} C_VEL
LIN {X 0,Y 452.462,Z 631.683,A -85,B 0,C 180,E1 -8369.999,E2 -8369.999} C_VEL
LIN {X 0,Y 452.454,Z 631.019,A -85,B 0,C 180,E1 -8371.779,E2 -8371.779} C_VEL
LIN {X 0,Y 452.474,Z 628.998,A -85,B 0,C 180,E1 -8373.561,E2 -8373.561} C_VEL
LIN {X 0,Y 452.552,Z 625.573,A -85,B 0,C 180,E1 -8375.346,E2 -8375.346} C_VEL
LIN {X 0,Y 452.653,Z 620.644,A -85,B 0,C 180,E1 -8377.134,E2 -8377.134} C_VEL
LIN {X 0,Y 452.893,Z 614.071,A -85,B 0,C 180,E1 -8378.926,E2 -8378.926} C_VEL
LIN {X 0,Y 453.219,Z 606.768,A -85,B 0,C 180,E1 -8380.497,E2 -8380.497} C_VEL
LIN {X 0,Y 453.695,Z 599.127,A -85,B 0,C 180,E1 -8381.843,E2 -8381.843} C_VEL
LIN {X 0,Y 454.258,Z 589.845,A -85,B 0,C 180,E1 -8383.21,E2 -8383.21} C_VEL
LIN {X 0,Y 454.923,Z 578.93,A -85,B 0,C 180,E1 -8384.538,E2 -8384.538} C_VEL
LIN {X 0,Y 455.753,Z 567.684,A -85,B 0,C 180,E1 -8385.655,E2 -8385.655} C_VEL
LIN {X 0,Y 456.567,Z 555.273,A -85,B 0,C 180,E1 -8386.659,E2 -8386.659} C_VEL
LIN {X 0,Y 457.367,Z 542.146,A -85,B 0,C 180,E1 -8387.504,E2 -8387.504} C_VEL
LIN {X 0,Y 457.963,Z 529.025,A -85,B 0,C 180,E1 -8388.162,E2 -8388.162} C_VEL
LIN {X 0,Y 458.598,Z 514.536,A -85,B 0,C 180,E1 -8388.685,E2 -8388.685} C_VEL
LIN {X 0,Y 459.015,Z 500.308,A -85,B 0,C 180,E1 -8389.015,E2 -8389.015} C_VEL
LIN {X 0,Y 460.252,Z 392.425,A -85,B 0,C 180,E1 -8390.746,E2 -8390.746} C_VEL
LIN {X 0,Y 455.926,Z 367.655,A -85,B 0,C 180,E1 -8391.387,E2 -8391.387} C_VEL
LIN {X 0,Y 456.789,Z 352.606,A -85,B 0,C 180,E1 -8393.819,E2 -8393.819} C_VEL
LIN {X 0,Y 457.488,Z 341.133,A -85,B 0,C 180,E1 -8395.719,E2 -8395.719} C_VEL
LIN {X 0,Y 455.549,Z 331.131,A -85,B 0,C 180,E1 -8397.568,E2 -8397.568} C_VEL
LIN {X 0,Y 453.521,Z 322.62,A -85,B 0,C 180,E1 -8399.217,E2 -8399.217} C_VEL
LIN {X 0,Y 453.48,Z 322.627,A -85,B 0,C 180,E1 -8402.848,E2 -8402.848} C_VEL
LIN {X 0,Y 453.454,Z 322.622,A -85,B 0,C 180,E1 -8406.082,E2 -8406.082} C_VEL
LIN {X 0,Y 453.526,Z 322.616,A -85,B 0,C 180,E1 -8409.445,E2 -8409.445} C_VEL
LIN {X 0,Y 453.459,Z 322.627,A -85,B 0,C 180,E1 -8412.994,E2 -8412.994} C_VEL
LIN {X 0,Y 453.468,Z 322.615,A -85,B 0,C 180,E1 -8415.779,E2 -8415.779} C_VEL
LIN {X 0,Y 453.476,Z 322.624,A -85,B 0,C 180,E1 -8418.209,E2 -8418.209} C_VEL
LIN {X 0,Y 453.489,Z 322.614,A -85,B 0,C 180,E1 -8420.792,E2 -8420.792} C_VEL
LIN {X 0,Y 453.451,Z 322.625,A -85,B 0,C 180,E1 -8423.917,E2 -8423.917} C_VEL
LIN {X 0,Y 453.477,Z 322.618,A -85,B 0,C 180,E1 -8427.15,E2 -8427.15} C_VEL
LIN {X 0,Y 453.508,Z 322.618,A -85,B 0,C 180,E1 -8430.27,E2 -8430.27} C_VEL
LIN {X 0,Y 453.504,Z 322.613,A -85,B 0,C 180,E1 -8433.294,E2 -8433.294} C_VEL
LIN {X 0,Y 453.494,Z 322.621,A -85,B 0,C 180,E1 -8436.238,E2 -8436.238} C_VEL
LIN {X 0,Y 453.474,Z 322.62,A -85,B 0,C 180,E1 -8439.117,E2 -8439.117} C_VEL
LIN {X 0,Y 453.504,Z 322.617,A -85,B 0,C 180,E1 -8441.944,E2 -8441.944} C_VEL
LIN {X 0,Y 453.541,Z 322.607,A -85,B 0,C 180,E1 -8444.726,E2 -8444.726} C_VEL
LIN {X 0,Y 453.55,Z 322.608,A -85,B 0,C 180,E1 -8448.378,E2 -8448.378} C_VEL
LIN {X 0,Y 453.643,Z 322.601,A -85,B 0,C 180,E1 -8451.985,E2 -8451.985} C_VEL
LIN {X 0,Y 453.655,Z 322.598,A -85,B 0,C 180,E1 -8454.666,E2 -8454.666} C_VEL
LIN {X 0,Y 453.677,Z 322.597,A -85,B 0,C 180,E1 -8458.224,E2 -8458.224} C_VEL
LIN {X 0,Y 453.757,Z 322.586,A -85,B 0,C 180,E1 -8460,E2 -8460} C_VEL
LIN {X 0,Y 453.721,Z 322.589,A -85,B 0,C 180,E1 -8462.663,E2 -8462.663} C_VEL
LIN {X 0,Y 453.618,Z 322.603,A -85,B 0,C 180,E1 -8466.226,E2 -8466.226} C_VEL
LIN {X 0,Y 453.55,Z 322.609,A -85,B 0,C 180,E1 -8468.914,E2 -8468.914} C_VEL
LIN {X 0,Y 453.554,Z 322.607,A -85,B 0,C 180,E1 -8472.529,E2 -8472.529} C_VEL
LIN {X 0,Y 453.527,Z 322.611,A -85,B 0,C 180,E1 -8476.196,E2 -8476.196} C_VEL
LIN {X 0,Y 453.507,Z 322.62,A -85,B 0,C 180,E1 -8479.039,E2 -8479.039} C_VEL
LIN {X 0,Y 453.465,Z 322.62,A -85,B 0,C 180,E1 -8481.836,E2 -8481.836} C_VEL
LIN {X 0,Y 453.483,Z 322.622,A -85,B 0,C 180,E1 -8484.736,E2 -8484.736} C_VEL
LIN {X 0,Y 453.465,Z 322.616,A -85,B 0,C 180,E1 -8487.946,E2 -8487.946} C_VEL
LIN {X 0,Y 453.464,Z 322.627,A -85,B 0,C 180,E1 -8490.76,E2 -8490.76} C_VEL
LIN {X 0,Y 453.458,Z 322.624,A -85,B 0,C 180,E1 -8493.914,E2 -8493.914} C_VEL
LIN {X 0,Y 453.443,Z 322.627,A -85,B 0,C 180,E1 -8497.19,E2 -8497.19} C_VEL
LIN {X 0,Y 453.474,Z 322.619,A -85,B 0,C 180,E1 -8499.451,E2 -8499.451} C_VEL
LIN {X 0,Y 453.467,Z 322.619,A -85,B 0,C 180,E1 -8501.935,E2 -8501.935} C_VEL
LIN {X 0,Y 453.476,Z 322.621,A -85,B 0,C 180,E1 -8505.472,E2 -8505.472} C_VEL
LIN {X 0,Y 453.503,Z 322.662,A -85,B 0,C 180,E1 -8507.553,E2 -8507.553} C_VEL
LIN {X 0,Y 455.975,Z 334.39,A -85,B 0,C 180,E1 -8510.147,E2 -8510.147} C_VEL
LIN {X 0,Y 456.236,Z 336.872,A -85,B 0,C 180,E1 -8510.67,E2 -8510.67} C_VEL
LIN {X 0,Y 460.559,Z 355.644,A -85,B 0,C 180,E1 -8511.228,E2 -8511.228} C_VEL
LIN {X 0,Y 459.134,Z 473.735,A -85,B 0,C 180,E1 -8513.15,E2 -8513.15} C_VEL
LIN {X 0,Y 458.728,Z 487.617,A -85,B 0,C 180,E1 -8513.549,E2 -8513.549} C_VEL
LIN {X 0,Y 458.242,Z 500.497,A -85,B 0,C 180,E1 -8514.083,E2 -8514.083} C_VEL
LIN {X 0,Y 457.6,Z 514.091,A -85,B 0,C 180,E1 -8514.836,E2 -8514.836} C_VEL
LIN {X 0,Y 456.835,Z 526.447,A -85,B 0,C 180,E1 -8515.707,E2 -8515.707} C_VEL
LIN {X 0,Y 456.066,Z 538.06,A -85,B 0,C 180,E1 -8516.723,E2 -8516.723} C_VEL
LIN {X 0,Y 455.43,Z 547.988,A -85,B 0,C 180,E1 -8517.774,E2 -8517.774} C_VEL
LIN {X 0,Y 454.698,Z 558.218,A -85,B 0,C 180,E1 -8519.076,E2 -8519.076} C_VEL
LIN {X 0,Y 454.567,Z 560.365,A -85,B 0,C 180,E1 -8519.38,E2 -8519.38} C_VEL
LIN {X 0,Y 453.633,Z 564.224,A -85,B 0,C 180,E1 -8519.943,E2 -8519.943} C_VEL
LIN {X 0,Y 450.401,Z 570.172,A -85,B 0,C 180,E1 -8520.862,E2 -8520.862} C_VEL
LIN {X 0,Y 447.206,Z 575.624,A -85,B 0,C 180,E1 -8521.835,E2 -8521.835} C_VEL
LIN {X 0,Y 446.332,Z 578.597,A -85,B 0,C 180,E1 -8522.476,E2 -8522.476} C_VEL
LIN {X 0,Y 445.959,Z 584.257,A -85,B 0,C 180,E1 -8523.932,E2 -8523.932} C_VEL
LIN {X 0,Y 445.666,Z 589.918,A -85,B 0,C 180,E1 -8525.796,E2 -8525.796} C_VEL
LIN {X 0,Y 445.545,Z 592.251,A -85,B 0,C 180,E1 -8526.776,E2 -8526.776} C_VEL
LIN {X 0,Y 445.392,Z 595.417,A -85,B 0,C 180,E1 -8528.587,E2 -8528.587} C_VEL
LIN {X 0,Y 445.303,Z 596.65,A -85,B 0,C 180,E1 -8529.684,E2 -8529.684} C_VEL
LIN {X 0,Y 445.313,Z 597.672,A -85,B 0,C 180,E1 -8531.601,E2 -8531.601} C_VEL
LIN {X 0,Y 445.262,Z 597.251,A -85,B 0,C 180,E1 -8533.495,E2 -8533.495} C_VEL
LIN {X 0,Y 445.365,Z 595.406,A -85,B 0,C 180,E1 -8535.376,E2 -8535.376} C_VEL
LIN {X 0,Y 445.536,Z 592.113,A -85,B 0,C 180,E1 -8537.243,E2 -8537.243} C_VEL
LIN {X 0,Y 445.766,Z 587.277,A -85,B 0,C 180,E1 -8539.095,E2 -8539.095} C_VEL
LIN {X 0,Y 445.994,Z 582.62,A -85,B 0,C 180,E1 -8540.477,E2 -8540.477} C_VEL
LIN {X 0,Y 446.399,Z 575.876,A -85,B 0,C 180,E1 -8542.076,E2 -8542.076} C_VEL
LIN {X 0,Y 446.958,Z 567.437,A -85,B 0,C 180,E1 -8543.682,E2 -8543.682} C_VEL
LIN {X 0,Y 447.518,Z 558.705,A -85,B 0,C 180,E1 -8545.046,E2 -8545.046} C_VEL
LIN {X 0,Y 448.259,Z 548.135,A -85,B 0,C 180,E1 -8546.405,E2 -8546.405} C_VEL
LIN {X 0,Y 448.999,Z 537.476,A -85,B 0,C 180,E1 -8547.534,E2 -8547.534} C_VEL
LIN {X 0,Y 449.73,Z 526.024,A -85,B 0,C 180,E1 -8548.533,E2 -8548.533} C_VEL
LIN {X 0,Y 450.507,Z 513.072,A -85,B 0,C 180,E1 -8549.442,E2 -8549.442} C_VEL
LIN {X 0,Y 451.188,Z 499.783,A -85,B 0,C 180,E1 -8550.168,E2 -8550.168} C_VEL
LIN {X 0,Y 451.651,Z 485.283,A -85,B 0,C 180,E1 -8550.753,E2 -8550.753} C_VEL
LIN {X 0,Y 452.035,Z 471.807,A -85,B 0,C 180,E1 -8551.114,E2 -8551.114} C_VEL
LIN {X 0,Y 453.301,Z 356.088,A -85,B 0,C 180,E1 -8552.996,E2 -8552.996} C_VEL
LIN {X 0,Y 449.039,Z 336.691,A -85,B 0,C 180,E1 -8553.54,E2 -8553.54} C_VEL
LIN {X 0,Y 446.602,Z 323.482,A -85,B 0,C 180,E1 -8556.353,E2 -8556.353} C_VEL
LIN {X 0,Y 446.528,Z 323.49,A -85,B 0,C 180,E1 -8559.056,E2 -8559.056} C_VEL
LIN {X 0,Y 446.52,Z 323.487,A -85,B 0,C 180,E1 -8562.73,E2 -8562.73} C_VEL
LIN {X 0,Y 446.487,Z 323.49,A -85,B 0,C 180,E1 -8566.46,E2 -8566.46} C_VEL
LIN {X 0,Y 446.467,Z 323.498,A -85,B 0,C 180,E1 -8569.304,E2 -8569.304} C_VEL
LIN {X 0,Y 446.415,Z 323.498,A -85,B 0,C 180,E1 -8572.2,E2 -8572.2} C_VEL
LIN {X 0,Y 446.418,Z 323.505,A -85,B 0,C 180,E1 -8575.155,E2 -8575.155} C_VEL
LIN {X 0,Y 446.415,Z 323.498,A -85,B 0,C 180,E1 -8578.184,E2 -8578.184} C_VEL
LIN {X 0,Y 446.388,Z 323.505,A -85,B 0,C 180,E1 -8581.303,E2 -8581.303} C_VEL
LIN {X 0,Y 446.412,Z 323.501,A -85,B 0,C 180,E1 -8584.525,E2 -8584.525} C_VEL
LIN {X 0,Y 446.395,Z 323.501,A -85,B 0,C 180,E1 -8588.077,E2 -8588.077} C_VEL
LIN {X 0,Y 446.399,Z 323.502,A -85,B 0,C 180,E1 -8591.395,E2 -8591.395} C_VEL
LIN {X 0,Y 446.42,Z 323.501,A -85,B 0,C 180,E1 -8595.108,E2 -8595.108} C_VEL
LIN {X 0,Y 446.396,Z 323.507,A -85,B 0,C 180,E1 -8598.606,E2 -8598.606} C_VEL
LIN {X 0,Y 446.387,Z 323.504,A -85,B 0,C 180,E1 -8602.12,E2 -8602.12} C_VEL
LIN {X 0,Y 446.419,Z 323.498,A -85,B 0,C 180,E1 -8605.477,E2 -8605.477} C_VEL
LIN {X 0,Y 446.409,Z 323.504,A -85,B 0,C 180,E1 -8608.7,E2 -8608.7} C_VEL
LIN {X 0,Y 446.424,Z 323.498,A -85,B 0,C 180,E1 -8611.837,E2 -8611.837} C_VEL
LIN {X 0,Y 446.421,Z 323.5,A -85,B 0,C 180,E1 -8614.846,E2 -8614.846} C_VEL
LIN {X 0,Y 446.447,Z 323.501,A -85,B 0,C 180,E1 -8618.247,E2 -8618.247} C_VEL
LIN {X 0,Y 446.441,Z 323.496,A -85,B 0,C 180,E1 -8621.649,E2 -8621.649} C_VEL
LIN {X 0,Y 446.461,Z 323.497,A -85,B 0,C 180,E1 -8624.478,E2 -8624.478} C_VEL
LIN {X 0,Y 446.519,Z 323.485,A -85,B 0,C 180,E1 -8627.384,E2 -8627.384} C_VEL
LIN {X 0,Y 446.533,Z 323.484,A -85,B 0,C 180,E1 -8630.945,E2 -8630.945} C_VEL
LIN {X 0,Y 446.618,Z 323.476,A -85,B 0,C 180,E1 -8633.676,E2 -8633.676} C_VEL
LIN {X 0,Y 446.684,Z 323.465,A -85,B 0,C 180,E1 -8637.295,E2 -8637.295} C_VEL
LIN {X 0,Y 446.79,Z 323.46,A -85,B 0,C 180,E1 -8640,E2 -8640} C_VEL
LIN {X 0,Y 446.681,Z 323.465,A -85,B 0,C 180,E1 -8642.706,E2 -8642.706} C_VEL
LIN {X 0,Y 446.622,Z 323.475,A -85,B 0,C 180,E1 -8646.324,E2 -8646.324} C_VEL
LIN {X 0,Y 446.54,Z 323.483,A -85,B 0,C 180,E1 -8649.056,E2 -8649.056} C_VEL
LIN {X 0,Y 446.525,Z 323.484,A -85,B 0,C 180,E1 -8652.73,E2 -8652.73} C_VEL
LIN {X 0,Y 446.494,Z 323.489,A -85,B 0,C 180,E1 -8656.459,E2 -8656.459} C_VEL
LIN {X 0,Y 446.473,Z 323.494,A -85,B 0,C 180,E1 -8659.303,E2 -8659.303} C_VEL
LIN {X 0,Y 446.421,Z 323.499,A -85,B 0,C 180,E1 -8662.2,E2 -8662.2} C_VEL
LIN {X 0,Y 446.448,Z 323.497,A -85,B 0,C 180,E1 -8665.153,E2 -8665.153} C_VEL
LIN {X 0,Y 446.489,Z 323.49,A -85,B 0,C 180,E1 -8668.179,E2 -8668.179} C_VEL
LIN {X 0,Y 446.423,Z 323.501,A -85,B 0,C 180,E1 -8671.775,E2 -8671.775} C_VEL
LIN {X 0,Y 446.432,Z 323.496,A -85,B 0,C 180,E1 -8674.523,E2 -8674.523} C_VEL
LIN {X 0,Y 446.417,Z 323.498,A -85,B 0,C 180,E1 -8678.079,E2 -8678.079} C_VEL
LIN {X 0,Y 446.431,Z 323.499,A -85,B 0,C 180,E1 -8680.917,E2 -8680.917} C_VEL
LIN {X 0,Y 446.426,Z 323.498,A -85,B 0,C 180,E1 -8683.843,E2 -8683.843} C_VEL
LIN {X 0,Y 446.403,Z 323.5,A -85,B 0,C 180,E1 -8686.403,E2 -8686.403} C_VEL
LIN {X 0,Y 446.431,Z 323.503,A -85,B 0,C 180,E1 -8689.082,E2 -8689.082} C_VEL
LIN {X 0,Y 446.413,Z 323.498,A -85,B 0,C 180,E1 -8692.121,E2 -8692.121} C_VEL
LIN {X 0,Y 446.433,Z 323.499,A -85,B 0,C 180,E1 -8695.477,E2 -8695.477} C_VEL
LIN {X 0,Y 446.42,Z 323.507,A -85,B 0,C 180,E1 -8698.699,E2 -8698.699} C_VEL
LIN {X 0,Y 446.49,Z 323.581,A -85,B 0,C 180,E1 -8700.94,E2 -8700.94} C_VEL
LIN {X 0,Y 449.946,Z 339.257,A -85,B 0,C 180,E1 -8703.82,E2 -8703.82} C_VEL
LIN {X 0,Y 450.273,Z 342.33,A -85,B 0,C 180,E1 -8704.355,E2 -8704.355} C_VEL
LIN {X 0,Y 449.137,Z 362.472,A -85,B 0,C 180,E1 -8707.66,E2 -8707.66} C_VEL
LIN {X 0,Y 448.787,Z 367.589,A -85,B 0,C 180,E1 -8708.488,E2 -8708.488} C_VEL
LIN {X 0,Y 453.171,Z 393.509,A -85,B 0,C 180,E1 -8709.117,E2 -8709.117} C_VEL
LIN {X 0,Y 451.797,Z 505.408,A -85,B 0,C 180,E1 -8710.933,E2 -8710.933} C_VEL
LIN {X 0,Y 451.3,Z 520.239,A -85,B 0,C 180,E1 -8711.353,E2 -8711.353} C_VEL
LIN {X 0,Y 450.721,Z 533.242,A -85,B 0,C 180,E1 -8711.89,E2 -8711.89} C_VEL
LIN {X 0,Y 450.051,Z 546.287,A -85,B 0,C 180,E1 -8712.607,E2 -8712.607} C_VEL
LIN {X 0,Y 449.222,Z 559.365,A -85,B 0,C 180,E1 -8713.526,E2 -8713.526} C_VEL
LIN {X 0,Y 448.434,Z 571.056,A -85,B 0,C 180,E1 -8714.547,E2 -8714.547} C_VEL
LIN {X 0,Y 447.685,Z 581.768,A -85,B 0,C 180,E1 -8715.684,E2 -8715.684} C_VEL
LIN {X 0,Y 447.043,Z 592.636,A -85,B 0,C 180,E1 -8717.087,E2 -8717.087} C_VEL
LIN {X 0,Y 446.446,Z 602.485,A -85,B 0,C 180,E1 -8718.651,E2 -8718.651} C_VEL
LIN {X 0,Y 445.945,Z 610.596,A -85,B 0,C 180,E1 -8720.245,E2 -8720.245} C_VEL
LIN {X 0,Y 445.643,Z 617.126,A -85,B 0,C 180,E1 -8721.839,E2 -8721.839} C_VEL
LIN {X 0,Y 445.5,Z 621.654,A -85,B 0,C 180,E1 -8723.204,E2 -8723.204} C_VEL
LIN {X 0,Y 445.459,Z 625.203,A -85,B 0,C 180,E1 -8724.567,E2 -8724.567} C_VEL
LIN {X 0,Y 445.375,Z 628.663,A -85,B 0,C 180,E1 -8726.38,E2 -8726.38} C_VEL
LIN {X 0,Y 445.43,Z 629.865,A -85,B 0,C 180,E1 -8727.286,E2 -8727.286} C_VEL
LIN {X 0,Y 445.364,Z 631.234,A -85,B 0,C 180,E1 -8729.095,E2 -8729.095} C_VEL
LIN {X 0,Y 445.364,Z 631.254,A -85,B 0,C 180,E1 -8730.903,E2 -8730.903} C_VEL
LIN {X 0,Y 445.429,Z 629.927,A -85,B 0,C 180,E1 -8732.712,E2 -8732.712} C_VEL
LIN {X 0,Y 445.395,Z 627.217,A -85,B 0,C 180,E1 -8734.524,E2 -8734.524} C_VEL
LIN {X 0,Y 445.528,Z 622.937,A -85,B 0,C 180,E1 -8736.385,E2 -8736.385} C_VEL
LIN {X 0,Y 445.649,Z 617.349,A -85,B 0,C 180,E1 -8738.159,E2 -8738.159} C_VEL
LIN {X 0,Y 445.981,Z 610.92,A -85,B 0,C 180,E1 -8739.752,E2 -8739.752} C_VEL
LIN {X 0,Y 446.463,Z 602.943,A -85,B 0,C 180,E1 -8741.347,E2 -8741.347} C_VEL
LIN {X 0,Y 447.013,Z 593.437,A -85,B 0,C 180,E1 -8742.897,E2 -8742.897} C_VEL
LIN {X 0,Y 447.631,Z 584.604,A -85,B 0,C 180,E1 -8744.084,E2 -8744.084} C_VEL
LIN {X 0,Y 448.439,Z 573.488,A -85,B 0,C 180,E1 -8745.334,E2 -8745.334} C_VEL
LIN {X 0,Y 449.364,Z 561.066,A -85,B 0,C 180,E1 -8746.467,E2 -8746.467} C_VEL
LIN {X 0,Y 450.193,Z 548.248,A -85,B 0,C 180,E1 -8747.405,E2 -8747.405} C_VEL
LIN {X 0,Y 451.017,Z 533.999,A -85,B 0,C 180,E1 -8748.216,E2 -8748.216} C_VEL
LIN {X 0,Y 451.663,Z 520.817,A -85,B 0,C 180,E1 -8748.777,E2 -8748.777} C_VEL
LIN {X 0,Y 452.172,Z 507.767,A -85,B 0,C 180,E1 -8749.167,E2 -8749.167} C_VEL
LIN {X 0,Y 452.567,Z 484.044,A -85,B 0,C 180,E1 -8749.592,E2 -8749.592} C_VEL
LIN {X 0,Y 453.607,Z 392.682,A -85,B 0,C 180,E1 -8751.085,E2 -8751.085} C_VEL
LIN {X 0,Y 449.435,Z 369.045,A -85,B 0,C 180,E1 -8751.715,E2 -8751.715} C_VEL
LIN {X 0,Y 449.088,Z 367.031,A -85,B 0,C 180,E1 -8751.794,E2 -8751.794} C_VEL
LIN {X 0,Y 450.336,Z 348.245,A -85,B 0,C 180,E1 -8754.92,E2 -8754.92} C_VEL
LIN {X 0,Y 450.64,Z 342.524,A -85,B 0,C 180,E1 -8755.891,E2 -8755.891} C_VEL
LIN {X 0,Y 448.303,Z 331.117,A -85,B 0,C 180,E1 -8758.053,E2 -8758.053} C_VEL
LIN {X 0,Y 446.463,Z 323.499,A -85,B 0,C 180,E1 -8759.585,E2 -8759.585} C_VEL
LIN {X 0,Y 446.42,Z 323.502,A -85,B 0,C 180,E1 -8762.36,E2 -8762.36} C_VEL
LIN {X 0,Y 446.418,Z 323.499,A -85,B 0,C 180,E1 -8765.625,E2 -8765.625} C_VEL
LIN {X 0,Y 446.469,Z 323.494,A -85,B 0,C 180,E1 -8769.023,E2 -8769.023} C_VEL
LIN {X 0,Y 446.431,Z 323.494,A -85,B 0,C 180,E1 -8772.277,E2 -8772.277} C_VEL
LIN {X 0,Y 446.451,Z 323.491,A -85,B 0,C 180,E1 -8775.102,E2 -8775.102} C_VEL
LIN {X 0,Y 446.424,Z 323.502,A -85,B 0,C 180,E1 -8778.608,E2 -8778.608} C_VEL
LIN {X 0,Y 446.44,Z 323.493,A -85,B 0,C 180,E1 -8780.972,E2 -8780.972} C_VEL
LIN {X 0,Y 446.415,Z 323.502,A -85,B 0,C 180,E1 -8784.373,E2 -8784.373} C_VEL
LIN {X 0,Y 446.416,Z 323.497,A -85,B 0,C 180,E1 -8787.638,E2 -8787.638} C_VEL
LIN {X 0,Y 446.463,Z 323.495,A -85,B 0,C 180,E1 -8790.791,E2 -8790.791} C_VEL
LIN {X 0,Y 446.471,Z 323.492,A -85,B 0,C 180,E1 -8793.848,E2 -8793.848} C_VEL
LIN {X 0,Y 446.42,Z 323.495,A -85,B 0,C 180,E1 -8796.823,E2 -8796.823} C_VEL
LIN {X 0,Y 446.436,Z 323.5,A -85,B 0,C 180,E1 -8799.736,E2 -8799.736} C_VEL
LIN {X 0,Y 446.457,Z 323.496,A -85,B 0,C 180,E1 -8802.597,E2 -8802.597} C_VEL
LIN {X 0,Y 446.464,Z 323.489,A -85,B 0,C 180,E1 -8805.412,E2 -8805.412} C_VEL
LIN {X 0,Y 446.508,Z 323.487,A -85,B 0,C 180,E1 -8808.193,E2 -8808.193} C_VEL
LIN {X 0,Y 446.591,Z 323.481,A -85,B 0,C 180,E1 -8811.857,E2 -8811.857} C_VEL
LIN {X 0,Y 446.63,Z 323.473,A -85,B 0,C 180,E1 -8814.582,E2 -8814.582} C_VEL
LIN {X 0,Y 446.647,Z 323.473,A -85,B 0,C 180,E1 -8818.196,E2 -8818.196} C_VEL
LIN {X 0,Y 446.708,Z 323.464,A -85,B 0,C 180,E1 -8820,E2 -8820} C_VEL
LIN {X 0,Y 446.668,Z 323.467,A -85,B 0,C 180,E1 -8822.705,E2 -8822.705} C_VEL
LIN {X 0,Y 446.588,Z 323.478,A -85,B 0,C 180,E1 -8826.324,E2 -8826.324} C_VEL
LIN {X 0,Y 446.501,Z 323.488,A -85,B 0,C 180,E1 -8829.056,E2 -8829.056} C_VEL
LIN {X 0,Y 446.511,Z 323.485,A -85,B 0,C 180,E1 -8832.73,E2 -8832.73} C_VEL
LIN {X 0,Y 446.473,Z 323.489,A -85,B 0,C 180,E1 -8836.459,E2 -8836.459} C_VEL
LIN {X 0,Y 446.458,Z 323.497,A -85,B 0,C 180,E1 -8839.303,E2 -8839.303} C_VEL
LIN {X 0,Y 446.406,Z 323.497,A -85,B 0,C 180,E1 -8842.2,E2 -8842.2} C_VEL
LIN {X 0,Y 446.428,Z 323.502,A -85,B 0,C 180,E1 -8845.154,E2 -8845.154} C_VEL
LIN {X 0,Y 446.428,Z 323.493,A -85,B 0,C 180,E1 -8848.182,E2 -8848.182} C_VEL
LIN {X 0,Y 446.405,Z 323.507,A -85,B 0,C 180,E1 -8851.301,E2 -8851.301} C_VEL
LIN {X 0,Y 446.413,Z 323.504,A -85,B 0,C 180,E1 -8854.524,E2 -8854.524} C_VEL
LIN {X 0,Y 446.404,Z 323.504,A -85,B 0,C 180,E1 -8858.079,E2 -8858.079} C_VEL
LIN {X 0,Y 446.418,Z 323.505,A -85,B 0,C 180,E1 -8860.918,E2 -8860.918} C_VEL
LIN {X 0,Y 446.389,Z 323.504,A -85,B 0,C 180,E1 -8863.847,E2 -8863.847} C_VEL
LIN {X 0,Y 446.421,Z 323.504,A -85,B 0,C 180,E1 -8866.78,E2 -8866.78} C_VEL
LIN {X 0,Y 446.464,Z 323.695,A -85,B 0,C 180,E1 -8867.263,E2 -8867.263} C_VEL
LIN {X 0,Y 449.128,Z 336.129,A -85,B 0,C 180,E1 -8870.063,E2 -8870.063} C_VEL
LIN {X 0,Y 449.33,Z 337.343,A -85,B 0,C 180,E1 -8870.303,E2 -8870.303} C_VEL
LIN {X 0,Y 452.875,Z 351.328,A -85,B 0,C 180,E1 -8870.744,E2 -8870.744} C_VEL
LIN {X 0,Y 454.006,Z 356.584,A -85,B 0,C 180,E1 -8870.895,E2 -8870.895} C_VEL
LIN {X 0,Y 452.513,Z 473.57,A -85,B 0,C 180,E1 -8872.826,E2 -8872.826} C_VEL
LIN {X 0,Y 452.073,Z 487.756,A -85,B 0,C 180,E1 -8873.237,E2 -8873.237} C_VEL
LIN {X 0,Y 451.54,Z 501.112,A -85,B 0,C 180,E1 -8873.801,E2 -8873.801} C_VEL
LIN {X 0,Y 450.866,Z 514.544,A -85,B 0,C 180,E1 -8874.561,E2 -8874.561} C_VEL
LIN {X 0,Y 450.011,Z 527.785,A -85,B 0,C 180,E1 -8875.521,E2 -8875.521} C_VEL
LIN {X 0,Y 449.202,Z 539.095,A -85,B 0,C 180,E1 -8876.539,E2 -8876.539} C_VEL
LIN {X 0,Y 448.414,Z 550.667,A -85,B 0,C 180,E1 -8877.815,E2 -8877.815} C_VEL
LIN {X 0,Y 447.688,Z 559.982,A -85,B 0,C 180,E1 -8879.063,E2 -8879.063} C_VEL
LIN {X 0,Y 446.971,Z 569.282,A -85,B 0,C 180,E1 -8880.571,E2 -8880.571} C_VEL
LIN {X 0,Y 446.455,Z 576.848,A -85,B 0,C 180,E1 -8882.076,E2 -8882.076} C_VEL
LIN {X 0,Y 446.332,Z 578.597,A -85,B 0,C 180,E1 -8882.476,E2 -8882.476} C_VEL
LIN {X 0,Y 445.478,Z 581.429,A -85,B 0,C 180,E1 -8883.133,E2 -8883.133} C_VEL
LIN {X 0,Y 442.381,Z 585.694,A -85,B 0,C 180,E1 -8884.218,E2 -8884.218} C_VEL
LIN {X 0,Y 439.325,Z 589.332,A -85,B 0,C 180,E1 -8885.352,E2 -8885.352} C_VEL
LIN {X 0,Y 438.551,Z 591.179,A -85,B 0,C 180,E1 -8886.08,E2 -8886.08} C_VEL
LIN {X 0,Y 438.377,Z 593.879,A -85,B 0,C 180,E1 -8887.372,E2 -8887.372} C_VEL
LIN {X 0,Y 438.331,Z 595.576,A -85,B 0,C 180,E1 -8888.425,E2 -8888.425} C_VEL
LIN {X 0,Y 438.186,Z 597.472,A -85,B 0,C 180,E1 -8890.318,E2 -8890.318} C_VEL
LIN {X 0,Y 438.221,Z 597.896,A -85,B 0,C 180,E1 -8891.293,E2 -8891.293} C_VEL
LIN {X 0,Y 438.174,Z 597.665,A -85,B 0,C 180,E1 -8893.22,E2 -8893.22} C_VEL
LIN {X 0,Y 438.28,Z 596.008,A -85,B 0,C 180,E1 -8895.135,E2 -8895.135} C_VEL
LIN {X 0,Y 438.427,Z 592.927,A -85,B 0,C 180,E1 -8897.032,E2 -8897.032} C_VEL
LIN {X 0,Y 438.678,Z 588.359,A -85,B 0,C 180,E1 -8898.917,E2 -8898.917} C_VEL
LIN {X 0,Y 438.879,Z 583.835,A -85,B 0,C 180,E1 -8900.321,E2 -8900.321} C_VEL
LIN {X 0,Y 439.31,Z 577.208,A -85,B 0,C 180,E1 -8901.977,E2 -8901.977} C_VEL
LIN {X 0,Y 439.81,Z 569.246,A -85,B 0,C 180,E1 -8903.578,E2 -8903.578} C_VEL
LIN {X 0,Y 440.45,Z 560.799,A -85,B 0,C 180,E1 -8904.966,E2 -8904.966} C_VEL
LIN {X 0,Y 441.249,Z 550.607,A -85,B 0,C 180,E1 -8906.348,E2 -8906.348} C_VEL
LIN {X 0,Y 441.938,Z 540.417,A -85,B 0,C 180,E1 -8907.494,E2 -8907.494} C_VEL
LIN {X 0,Y 442.804,Z 528.053,A -85,B 0,C 180,E1 -8908.627,E2 -8908.627} C_VEL
LIN {X 0,Y 443.586,Z 515.57,A -85,B 0,C 180,E1 -8909.547,E2 -8909.547} C_VEL
LIN {X 0,Y 444.338,Z 501.767,A -85,B 0,C 180,E1 -8910.341,E2 -8910.341} C_VEL
LIN {X 0,Y 444.824,Z 488.708,A -85,B 0,C 180,E1 -8910.906,E2 -8910.906} C_VEL
LIN {X 0,Y 445.202,Z 474.679,A -85,B 0,C 180,E1 -8911.329,E2 -8911.329} C_VEL
LIN {X 0,Y 445.757,Z 435.952,A -85,B 0,C 180,E1 -8911.991,E2 -8911.991} C_VEL
LIN {X 0,Y 446.643,Z 357.292,A -85,B 0,C 180,E1 -8913.281,E2 -8913.281} C_VEL
LIN {X 0,Y 442.333,Z 338.366,A -85,B 0,C 180,E1 -8913.804,E2 -8913.804} C_VEL
LIN {X 0,Y 441.975,Z 337.007,A -85,B 0,C 180,E1 -8913.853,E2 -8913.853} C_VEL
LIN {X 0,Y 439.568,Z 324.357,A -85,B 0,C 180,E1 -8916.623,E2 -8916.623} C_VEL
LIN {X 0,Y 439.455,Z 324.371,A -85,B 0,C 180,E1 -8920.133,E2 -8920.133} C_VEL
LIN {X 0,Y 439.463,Z 324.368,A -85,B 0,C 180,E1 -8922.938,E2 -8922.938} C_VEL
LIN {X 0,Y 439.445,Z 324.367,A -85,B 0,C 180,E1 -8926.349,E2 -8926.349} C_VEL
LIN {X 0,Y 439.401,Z 324.374,A -85,B 0,C 180,E1 -8929.627,E2 -8929.627} C_VEL
LIN {X 0,Y 439.361,Z 324.379,A -85,B 0,C 180,E1 -8932.576,E2 -8932.576} C_VEL
LIN {X 0,Y 439.364,Z 324.378,A -85,B 0,C 180,E1 -8935.588,E2 -8935.588} C_VEL
LIN {X 0,Y 439.379,Z 324.378,A -85,B 0,C 180,E1 -8938.677,E2 -8938.677} C_VEL
LIN {X 0,Y 439.341,Z 324.379,A -85,B 0,C 180,E1 -8942.025,E2 -8942.025} C_VEL
LIN {X 0,Y 439.383,Z 324.377,A -85,B 0,C 180,E1 -8945.339,E2 -8945.339} C_VEL
LIN {X 0,Y 439.352,Z 324.382,A -85,B 0,C 180,E1 -8948.599,E2 -8948.599} C_VEL
LIN {X 0,Y 439.362,Z 324.379,A -85,B 0,C 180,E1 -8951.253,E2 -8951.253} C_VEL
LIN {X 0,Y 439.395,Z 324.38,A -85,B 0,C 180,E1 -8954.731,E2 -8954.731} C_VEL
LIN {X 0,Y 439.345,Z 324.379,A -85,B 0,C 180,E1 -8957.79,E2 -8957.79} C_VEL
LIN {X 0,Y 439.348,Z 324.379,A -85,B 0,C 180,E1 -8961.402,E2 -8961.402} C_VEL
LIN {X 0,Y 439.391,Z 324.378,A -85,B 0,C 180,E1 -8964.844,E2 -8964.844} C_VEL
LIN {X 0,Y 439.369,Z 324.379,A -85,B 0,C 180,E1 -8968.14,E2 -8968.14} C_VEL
LIN {X 0,Y 439.387,Z 324.374,A -85,B 0,C 180,E1 -8971.61,E2 -8971.61} C_VEL
LIN {X 0,Y 439.367,Z 324.384,A -85,B 0,C 180,E1 -8974.413,E2 -8974.413} C_VEL
LIN {X 0,Y 439.355,Z 324.378,A -85,B 0,C 180,E1 -8977.424,E2 -8977.424} C_VEL
LIN {X 0,Y 439.442,Z 324.37,A -85,B 0,C 180,E1 -8980.664,E2 -8980.664} C_VEL
LIN {X 0,Y 439.421,Z 324.377,A -85,B 0,C 180,E1 -8984.223,E2 -8984.223} C_VEL
LIN {X 0,Y 439.487,Z 324.361,A -85,B 0,C 180,E1 -8987.286,E2 -8987.286} C_VEL
LIN {X 0,Y 439.497,Z 324.361,A -85,B 0,C 180,E1 -8990.799,E2 -8990.799} C_VEL
LIN {X 0,Y 439.569,Z 324.353,A -85,B 0,C 180,E1 -8993.574,E2 -8993.574} C_VEL
LIN {X 0,Y 439.425,Z 324.37,A -85,B 0,C 180,E1 -8995.414,E2 -8995.414} C_VEL
LIN {X 0,Y 439.635,Z 324.349,A -85,B 0,C 180,E1 -8998.168,E2 -8998.168} C_VEL
LIN {X 0,Y 439.759,Z 324.335,A -85,B 0,C 180,E1 -9000,E2 -9000} C_VEL
LIN {X 0,Y 439.63,Z 324.344,A -85,B 0,C 180,E1 -9002.749,E2 -9002.749} C_VEL
LIN {X 0,Y 439.594,Z 324.35,A -85,B 0,C 180,E1 -9006.426,E2 -9006.426} C_VEL
LIN {X 0,Y 439.502,Z 324.36,A -85,B 0,C 180,E1 -9009.202,E2 -9009.202} C_VEL
LIN {X 0,Y 439.469,Z 324.364,A -85,B 0,C 180,E1 -9012.938,E2 -9012.938} C_VEL
LIN {X 0,Y 439.451,Z 324.367,A -85,B 0,C 180,E1 -9016.349,E2 -9016.349} C_VEL
LIN {X 0,Y 439.407,Z 324.379,A -85,B 0,C 180,E1 -9019.626,E2 -9019.626} C_VEL
LIN {X 0,Y 439.368,Z 324.376,A -85,B 0,C 180,E1 -9022.576,E2 -9022.576} C_VEL
LIN {X 0,Y 439.402,Z 324.379,A -85,B 0,C 180,E1 -9025.585,E2 -9025.585} C_VEL
LIN {X 0,Y 439.421,Z 324.37,A -85,B 0,C 180,E1 -9028.673,E2 -9028.673} C_VEL
LIN {X 0,Y 439.374,Z 324.377,A -85,B 0,C 180,E1 -9032.03,E2 -9032.03} C_VEL
LIN {X 0,Y 439.397,Z 324.38,A -85,B 0,C 180,E1 -9035.34,E2 -9035.34} C_VEL
LIN {X 0,Y 439.386,Z 324.374,A -85,B 0,C 180,E1 -9038.595,E2 -9038.595} C_VEL
LIN {X 0,Y 439.392,Z 324.38,A -85,B 0,C 180,E1 -9041.257,E2 -9041.257} C_VEL
LIN {X 0,Y 439.409,Z 324.373,A -85,B 0,C 180,E1 -9044.729,E2 -9044.729} C_VEL
LIN {X 0,Y 439.4,Z 324.373,A -85,B 0,C 180,E1 -9047.795,E2 -9047.795} C_VEL
LIN {X 0,Y 439.43,Z 324.368,A -85,B 0,C 180,E1 -9050.227,E2 -9050.227} C_VEL
LIN {X 0,Y 439.378,Z 324.376,A -85,B 0,C 180,E1 -9053.713,E2 -9053.713} C_VEL
LIN {X 0,Y 439.377,Z 324.383,A -85,B 0,C 180,E1 -9057.054,E2 -9057.054} C_VEL
LIN {X 0,Y 439.447,Z 324.448,A -85,B 0,C 180,E1 -9060.673,E2 -9060.673} C_VEL
LIN {X 0,Y 442.938,Z 340.233,A -85,B 0,C 180,E1 -9063.623,E2 -9063.623} C_VEL
LIN {X 0,Y 443.301,Z 344.688,A -85,B 0,C 180,E1 -9064.404,E2 -9064.404} C_VEL
LIN {X 0,Y 442.066,Z 365.183,A -85,B 0,C 180,E1 -9067.816,E2 -9067.816} C_VEL
LIN {X 0,Y 441.913,Z 367.316,A -85,B 0,C 180,E1 -9068.166,E2 -9068.166} C_VEL
LIN {X 0,Y 446.437,Z 394.203,A -85,B 0,C 180,E1 -9068.832,E2 -9068.832} C_VEL
LIN {X 0,Y 445.029,Z 505.393,A -85,B 0,C 180,E1 -9070.661,E2 -9070.661} C_VEL
LIN {X 0,Y 444.523,Z 520.133,A -85,B 0,C 180,E1 -9071.088,E2 -9071.088} C_VEL
LIN {X 0,Y 443.935,Z 532.718,A -85,B 0,C 180,E1 -9071.613,E2 -9071.613} C_VEL
LIN {X 0,Y 443.2,Z 545.982,A -85,B 0,C 180,E1 -9072.351,E2 -9072.351} C_VEL
LIN {X 0,Y 442.357,Z 558.814,A -85,B 0,C 180,E1 -9073.263,E2 -9073.263} C_VEL
LIN {X 0,Y 441.523,Z 570.554,A -85,B 0,C 180,E1 -9074.299,E2 -9074.299} C_VEL
LIN {X 0,Y 440.739,Z 581.307,A -85,B 0,C 180,E1 -9075.454,E2 -9075.454} C_VEL
LIN {X 0,Y 440.052,Z 592.136,A -85,B 0,C 180,E1 -9076.868,E2 -9076.868} C_VEL
LIN {X 0,Y 439.484,Z 600.764,A -85,B 0,C 180,E1 -9078.235,E2 -9078.235} C_VEL
LIN {X 0,Y 438.927,Z 609.194,A -85,B 0,C 180,E1 -9079.855,E2 -9079.855} C_VEL
LIN {X 0,Y 438.664,Z 615.064,A -85,B 0,C 180,E1 -9081.245,E2 -9081.245} C_VEL
LIN {X 0,Y 438.491,Z 619.898,A -85,B 0,C 180,E1 -9082.632,E2 -9082.632} C_VEL
LIN {X 0,Y 438.356,Z 624.891,A -85,B 0,C 180,E1 -9084.479,E2 -9084.479} C_VEL
LIN {X 0,Y 438.276,Z 628.367,A -85,B 0,C 180,E1 -9086.322,E2 -9086.322} C_VEL
LIN {X 0,Y 438.356,Z 629.576,A -85,B 0,C 180,E1 -9087.242,E2 -9087.242} C_VEL
LIN {X 0,Y 438.276,Z 630.957,A -85,B 0,C 180,E1 -9089.08,E2 -9089.08} C_VEL
LIN {X 0,Y 438.276,Z 630.99,A -85,B 0,C 180,E1 -9090.918,E2 -9090.918} C_VEL
LIN {X 0,Y 438.337,Z 629.677,A -85,B 0,C 180,E1 -9092.756,E2 -9092.756} C_VEL
LIN {X 0,Y 438.319,Z 626.982,A -85,B 0,C 180,E1 -9094.597,E2 -9094.597} C_VEL
LIN {X 0,Y 438.447,Z 622.846,A -85,B 0,C 180,E1 -9096.442,E2 -9096.442} C_VEL
LIN {X 0,Y 438.593,Z 617.145,A -85,B 0,C 180,E1 -9098.291,E2 -9098.291} C_VEL
LIN {X 0,Y 438.906,Z 610.731,A -85,B 0,C 180,E1 -9099.911,E2 -9099.911} C_VEL
LIN {X 0,Y 439.465,Z 602.773,A -85,B 0,C 180,E1 -9101.53,E2 -9101.53} C_VEL
LIN {X 0,Y 440.013,Z 593.86,A -85,B 0,C 180,E1 -9103.015,E2 -9103.015} C_VEL
LIN {X 0,Y 440.713,Z 584.48,A -85,B 0,C 180,E1 -9104.31,E2 -9104.31} C_VEL
LIN {X 0,Y 441.486,Z 574.487,A -85,B 0,C 180,E1 -9105.464,E2 -9105.464} C_VEL
LIN {X 0,Y 442.418,Z 562.442,A -85,B 0,C 180,E1 -9106.614,E2 -9106.614} C_VEL
LIN {X 0,Y 443.359,Z 549.598,A -85,B 0,C 180,E1 -9107.599,E2 -9107.599} C_VEL
LIN {X 0,Y 444.133,Z 537.3,A -85,B 0,C 180,E1 -9108.347,E2 -9108.347} C_VEL
LIN {X 0,Y 444.822,Z 523.534,A -85,B 0,C 180,E1 -9108.987,E2 -9108.987} C_VEL
LIN {X 0,Y 445.468,Z 509.695,A -85,B 0,C 180,E1 -9109.437,E2 -9109.437} C_VEL
LIN {X 0,Y 445.831,Z 492.483,A -85,B 0,C 180,E1 -9109.78,E2 -9109.78} C_VEL
LIN {X 0,Y 447.071,Z 393.822,A -85,B 0,C 180,E1 -9111.413,E2 -9111.413} C_VEL
LIN {X 0,Y 442.983,Z 370.572,A -85,B 0,C 180,E1 -9112.049,E2 -9112.049} C_VEL
LIN {X 0,Y 442.279,Z 366.741,A -85,B 0,C 180,E1 -9112.181,E2 -9112.181} C_VEL
LIN {X 0,Y 443.602,Z 347.565,A -85,B 0,C 180,E1 -9115.437,E2 -9115.437} C_VEL
LIN {X 0,Y 443.769,Z 343.93,A -85,B 0,C 180,E1 -9116.069,E2 -9116.069} C_VEL
LIN {X 0,Y 441.397,Z 332.565,A -85,B 0,C 180,E1 -9118.273,E2 -9118.273} C_VEL
LIN {X 0,Y 439.396,Z 324.377,A -85,B 0,C 180,E1 -9119.954,E2 -9119.954} C_VEL
LIN {X 0,Y 439.37,Z 324.383,A -85,B 0,C 180,E1 -9122.945,E2 -9122.945} C_VEL
LIN {X 0,Y 439.374,Z 324.375,A -85,B 0,C 180,E1 -9126.286,E2 -9126.286} C_VEL
LIN {X 0,Y 439.423,Z 324.372,A -85,B 0,C 180,E1 -9129.852,E2 -9129.852} C_VEL
LIN {X 0,Y 439.378,Z 324.375,A -85,B 0,C 180,E1 -9132.626,E2 -9132.626} C_VEL
LIN {X 0,Y 439.401,Z 324.368,A -85,B 0,C 180,E1 -9135.27,E2 -9135.27} C_VEL
LIN {X 0,Y 439.384,Z 324.376,A -85,B 0,C 180,E1 -9138.742,E2 -9138.742} C_VEL
LIN {X 0,Y 439.377,Z 324.373,A -85,B 0,C 180,E1 -9141.605,E2 -9141.605} C_VEL
LIN {X 0,Y 439.395,Z 324.378,A -85,B 0,C 180,E1 -9144.843,E2 -9144.843} C_VEL
LIN {X 0,Y 439.369,Z 324.379,A -85,B 0,C 180,E1 -9148.139,E2 -9148.139} C_VEL
LIN {X 0,Y 439.419,Z 324.37,A -85,B 0,C 180,E1 -9151.326,E2 -9151.326} C_VEL
LIN {X 0,Y 439.394,Z 324.378,A -85,B 0,C 180,E1 -9154.414,E2 -9154.414} C_VEL
LIN {X 0,Y 439.357,Z 324.374,A -85,B 0,C 180,E1 -9157.424,E2 -9157.424} C_VEL
LIN {X 0,Y 439.434,Z 324.366,A -85,B 0,C 180,E1 -9160.662,E2 -9160.662} C_VEL
LIN {X 0,Y 439.467,Z 324.364,A -85,B 0,C 180,E1 -9164.224,E2 -9164.224} C_VEL
LIN {X 0,Y 439.474,Z 324.366,A -85,B 0,C 180,E1 -9168.001,E2 -9168.001} C_VEL
LIN {X 0,Y 439.539,Z 324.362,A -85,B 0,C 180,E1 -9171.726,E2 -9171.726} C_VEL
LIN {X 0,Y 439.605,Z 324.349,A -85,B 0,C 180,E1 -9174.495,E2 -9174.495} C_VEL
LIN {X 0,Y 439.617,Z 324.349,A -85,B 0,C 180,E1 -9178.167,E2 -9178.167} C_VEL
LIN {X 0,Y 439.659,Z 324.342,A -85,B 0,C 180,E1 -9180,E2 -9180} C_VEL
LIN {X 0,Y 439.618,Z 324.346,A -85,B 0,C 180,E1 -9182.749,E2 -9182.749} C_VEL
LIN {X 0,Y 439.54,Z 324.356,A -85,B 0,C 180,E1 -9186.426,E2 -9186.426} C_VEL
LIN {X 0,Y 439.467,Z 324.365,A -85,B 0,C 180,E1 -9189.202,E2 -9189.202} C_VEL
LIN {X 0,Y 439.454,Z 324.365,A -85,B 0,C 180,E1 -9192.938,E2 -9192.938} C_VEL
LIN {X 0,Y 439.434,Z 324.366,A -85,B 0,C 180,E1 -9196.347,E2 -9196.347} C_VEL
LIN {X 0,Y 439.391,Z 324.377,A -85,B 0,C 180,E1 -9199.626,E2 -9199.626} C_VEL
LIN {X 0,Y 439.352,Z 324.377,A -85,B 0,C 180,E1 -9202.576,E2 -9202.576} C_VEL
LIN {X 0,Y 439.367,Z 324.382,A -85,B 0,C 180,E1 -9205.587,E2 -9205.587} C_VEL
LIN {X 0,Y 439.381,Z 324.37,A -85,B 0,C 180,E1 -9208.676,E2 -9208.676} C_VEL
LIN {X 0,Y 439.358,Z 324.38,A -85,B 0,C 180,E1 -9212.03,E2 -9212.03} C_VEL
LIN {X 0,Y 439.382,Z 324.38,A -85,B 0,C 180,E1 -9215.34,E2 -9215.34} C_VEL
LIN {X 0,Y 439.366,Z 324.384,A -85,B 0,C 180,E1 -9218.596,E2 -9218.596} C_VEL
LIN {X 0,Y 439.38,Z 324.377,A -85,B 0,C 180,E1 -9221.257,E2 -9221.257} C_VEL
LIN {X 0,Y 439.391,Z 324.379,A -85,B 0,C 180,E1 -9224.73,E2 -9224.73} C_VEL
LIN {X 0,Y 439.418,Z 324.529,A -85,B 0,C 180,E1 -9226.911,E2 -9226.911} C_VEL
LIN {X 0,Y 442.152,Z 337.212,A -85,B 0,C 180,E1 -9229.826,E2 -9229.826} C_VEL
LIN {X 0,Y 442.288,Z 337.807,A -85,B 0,C 180,E1 -9229.907,E2 -9229.907} C_VEL
LIN {X 0,Y 444.839,Z 345.835,A -85,B 0,C 180,E1 -9230.197,E2 -9230.197} C_VEL
LIN {X 0,Y 447.521,Z 358.401,A -85,B 0,C 180,E1 -9230.57,E2 -9230.57} C_VEL
LIN {X 0,Y 445.898,Z 473.781,A -85,B 0,C 180,E1 -9232.5,E2 -9232.5} C_VEL
LIN {X 0,Y 445.46,Z 488.012,A -85,B 0,C 180,E1 -9232.918,E2 -9232.918} C_VEL
LIN {X 0,Y 444.895,Z 501.293,A -85,B 0,C 180,E1 -9233.486,E2 -9233.486} C_VEL
LIN {X 0,Y 444.244,Z 513.507,A -85,B 0,C 180,E1 -9234.174,E2 -9234.174} C_VEL
LIN {X 0,Y 443.411,Z 526.065,A -85,B 0,C 180,E1 -9235.071,E2 -9235.071} C_VEL
LIN {X 0,Y 442.597,Z 537.021,A -85,B 0,C 180,E1 -9236.036,E2 -9236.036} C_VEL
LIN {X 0,Y 441.754,Z 548.354,A -85,B 0,C 180,E1 -9237.255,E2 -9237.255} C_VEL
LIN {X 0,Y 440.93,Z 558.183,A -85,B 0,C 180,E1 -9238.535,E2 -9238.535} C_VEL
LIN {X 0,Y 440.172,Z 567.952,A -85,B 0,C 180,E1 -9240.084,E2 -9240.084} C_VEL
LIN {X 0,Y 439.566,Z 575.599,A -85,B 0,C 180,E1 -9241.565,E2 -9241.565} C_VEL
LIN {X 0,Y 439.159,Z 581.17,A -85,B 0,C 180,E1 -9242.866,E2 -9242.866} C_VEL
LIN {X 0,Y 438.798,Z 586.509,A -85,B 0,C 180,E1 -9244.378,E2 -9244.378} C_VEL
LIN {X 0,Y 438.551,Z 591.179,A -85,B 0,C 180,E1 -9246.08,E2 -9246.08} C_VEL
LIN {X 0,Y 437.786,Z 592.859,A -85,B 0,C 180,E1 -9246.815,E2 -9246.815} C_VEL
LIN {X 0,Y 434.797,Z 595.208,A -85,B 0,C 180,E1 -9248.019,E2 -9248.019} C_VEL
LIN {X 0,Y 432.303,Z 596.657,A -85,B 0,C 180,E1 -9249.001,E2 -9249.001} C_VEL
LIN {X 0,Y 431.22,Z 597.4,A -85,B 0,C 180,E1 -9249.769,E2 -9249.769} C_VEL
LIN {X 0,Y 431.124,Z 597.568,A -85,B 0,C 180,E1 -9250.031,E2 -9250.031} C_VEL
LIN {X 0,Y 431.09,Z 598.273,A -85,B 0,C 180,E1 -9251.957,E2 -9251.957} C_VEL
LIN {X 0,Y 431.117,Z 597.523,A -85,B 0,C 180,E1 -9253.912,E2 -9253.912} C_VEL
LIN {X 0,Y 431.194,Z 595.35,A -85,B 0,C 180,E1 -9255.85,E2 -9255.85} C_VEL
LIN {X 0,Y 431.432,Z 591.689,A -85,B 0,C 180,E1 -9257.792,E2 -9257.792} C_VEL
LIN {X 0,Y 431.677,Z 586.594,A -85,B 0,C 180,E1 -9259.684,E2 -9259.684} C_VEL
LIN {X 0,Y 432.02,Z 581.609,A -85,B 0,C 180,E1 -9261.111,E2 -9261.111} C_VEL
LIN {X 0,Y 432.487,Z 574.746,A -85,B 0,C 180,E1 -9262.708,E2 -9262.708} C_VEL
LIN {X 0,Y 433.062,Z 567.009,A -85,B 0,C 180,E1 -9264.179,E2 -9264.179} C_VEL
LIN {X 0,Y 433.685,Z 558.08,A -85,B 0,C 180,E1 -9265.586,E2 -9265.586} C_VEL
LIN {X 0,Y 434.397,Z 549.2,A -85,B 0,C 180,E1 -9266.755,E2 -9266.755} C_VEL
LIN {X 0,Y 435.174,Z 538.643,A -85,B 0,C 180,E1 -9267.918,E2 -9267.918} C_VEL
LIN {X 0,Y 436.002,Z 527.268,A -85,B 0,C 180,E1 -9268.95,E2 -9268.95} C_VEL
LIN {X 0,Y 436.809,Z 514.513,A -85,B 0,C 180,E1 -9269.886,E2 -9269.886} C_VEL
LIN {X 0,Y 437.555,Z 501.448,A -85,B 0,C 180,E1 -9270.634,E2 -9270.634} C_VEL
LIN {X 0,Y 438.068,Z 487.462,A -85,B 0,C 180,E1 -9271.236,E2 -9271.236} C_VEL
LIN {X 0,Y 438.512,Z 473.697,A -85,B 0,C 180,E1 -9271.637,E2 -9271.637} C_VEL
LIN {X 0,Y 439.963,Z 358.19,A -85,B 0,C 180,E1 -9273.576,E2 -9273.576} C_VEL
LIN {X 0,Y 435.711,Z 339.844,A -85,B 0,C 180,E1 -9274.096,E2 -9274.096} C_VEL
LIN {X 0,Y 434.769,Z 337.256,A -85,B 0,C 180,E1 -9274.202,E2 -9274.202} C_VEL
LIN {X 0,Y 432.524,Z 325.233,A -85,B 0,C 180,E1 -9276.846,E2 -9276.846} C_VEL
LIN {X 0,Y 432.4,Z 325.249,A -85,B 0,C 180,E1 -9280.3,E2 -9280.3} C_VEL
LIN {X 0,Y 432.398,Z 325.25,A -85,B 0,C 180,E1 -9283.154,E2 -9283.154} C_VEL
LIN {X 0,Y 432.41,Z 325.243,A -85,B 0,C 180,E1 -9286.479,E2 -9286.479} C_VEL
LIN {X 0,Y 432.337,Z 325.252,A -85,B 0,C 180,E1 -9289.961,E2 -9289.961} C_VEL
LIN {X 0,Y 432.309,Z 325.261,A -85,B 0,C 180,E1 -9292.966,E2 -9292.966} C_VEL
LIN {X 0,Y 432.315,Z 325.255,A -85,B 0,C 180,E1 -9296.036,E2 -9296.036} C_VEL
LIN {X 0,Y 432.319,Z 325.259,A -85,B 0,C 180,E1 -9299.19,E2 -9299.19} C_VEL
LIN {X 0,Y 432.303,Z 325.258,A -85,B 0,C 180,E1 -9302.445,E2 -9302.445} C_VEL
LIN {X 0,Y 432.33,Z 325.253,A -85,B 0,C 180,E1 -9305.819,E2 -9305.819} C_VEL
LIN {X 0,Y 432.299,Z 325.259,A -85,B 0,C 180,E1 -9309.349,E2 -9309.349} C_VEL
LIN {X 0,Y 432.301,Z 325.256,A -85,B 0,C 180,E1 -9311.802,E2 -9311.802} C_VEL
LIN {X 0,Y 432.333,Z 325.255,A -85,B 0,C 180,E1 -9314.348,E2 -9314.348} C_VEL
LIN {X 0,Y 432.3,Z 325.26,A -85,B 0,C 180,E1 -9317.019,E2 -9317.019} C_VEL
LIN {X 0,Y 432.287,Z 325.258,A -85,B 0,C 180,E1 -9319.829,E2 -9319.829} C_VEL
LIN {X 0,Y 432.294,Z 325.26,A -85,B 0,C 180,E1 -9323.021,E2 -9323.021} C_VEL
LIN {X 0,Y 432.332,Z 325.254,A -85,B 0,C 180,E1 -9326.003,E2 -9326.003} C_VEL
LIN {X 0,Y 432.341,Z 325.251,A -85,B 0,C 180,E1 -9329.492,E2 -9329.492} C_VEL
LIN {X 0,Y 432.32,Z 325.255,A -85,B 0,C 180,E1 -9331.873,E2 -9331.873} C_VEL
LIN {X 0,Y 432.324,Z 325.255,A -85,B 0,C 180,E1 -9334.997,E2 -9334.997} C_VEL
LIN {X 0,Y 432.354,Z 325.254,A -85,B 0,C 180,E1 -9338.046,E2 -9338.046} C_VEL
LIN {X 0,Y 432.382,Z 325.247,A -85,B 0,C 180,E1 -9341.03,E2 -9341.03} C_VEL
LIN {X 0,Y 432.39,Z 325.249,A -85,B 0,C 180,E1 -9343.96,E2 -9343.96} C_VEL
LIN {X 0,Y 432.461,Z 325.239,A -85,B 0,C 180,E1 -9347.804,E2 -9347.804} C_VEL
LIN {X 0,Y 432.466,Z 325.237,A -85,B 0,C 180,E1 -9351.59,E2 -9351.59} C_VEL
LIN {X 0,Y 432.582,Z 325.225,A -85,B 0,C 180,E1 -9354.406,E2 -9354.406} C_VEL
LIN {X 0,Y 432.605,Z 325.225,A -85,B 0,C 180,E1 -9358.138,E2 -9358.138} C_VEL
LIN {X 0,Y 432.728,Z 325.211,A -85,B 0,C 180,E1 -9360,E2 -9360} C_VEL
LIN {X 0,Y 432.582,Z 325.222,A -85,B 0,C 180,E1 -9362.794,E2 -9362.794} C_VEL
LIN {X 0,Y 432.588,Z 325.224,A -85,B 0,C 180,E1 -9365.594,E2 -9365.594} C_VEL
LIN {X 0,Y 432.486,Z 325.235,A -85,B 0,C 180,E1 -9368.41,E2 -9368.41} C_VEL
LIN {X 0,Y 432.463,Z 325.239,A -85,B 0,C 180,E1 -9372.197,E2 -9372.197} C_VEL
LIN {X 0,Y 432.434,Z 325.243,A -85,B 0,C 180,E1 -9376.039,E2 -9376.039} C_VEL
LIN {X 0,Y 432.391,Z 325.25,A -85,B 0,C 180,E1 -9379.485,E2 -9379.485} C_VEL
LIN {X 0,Y 432.322,Z 325.255,A -85,B 0,C 180,E1 -9382.964,E2 -9382.964} C_VEL
LIN {X 0,Y 432.365,Z 325.251,A -85,B 0,C 180,E1 -9386.033,E2 -9386.033} C_VEL
LIN {X 0,Y 432.347,Z 325.254,A -85,B 0,C 180,E1 -9389.187,E2 -9389.187} C_VEL
LIN {X 0,Y 432.327,Z 325.253,A -85,B 0,C 180,E1 -9392.443,E2 -9392.443} C_VEL
LIN {X 0,Y 432.347,Z 325.255,A -85,B 0,C 180,E1 -9395.632,E2 -9395.632} C_VEL
LIN {X 0,Y 432.354,Z 325.258,A -85,B 0,C 180,E1 -9399.343,E2 -9399.343} C_VEL
LIN {X 0,Y 432.338,Z 325.254,A -85,B 0,C 180,E1 -9401.797,E2 -9401.797} C_VEL
LIN {X 0,Y 432.344,Z 325.251,A -85,B 0,C 180,E1 -9404.346,E2 -9404.346} C_VEL
LIN {X 0,Y 432.324,Z 325.259,A -85,B 0,C 180,E1 -9407.015,E2 -9407.015} C_VEL
LIN {X 0,Y 432.337,Z 325.253,A -85,B 0,C 180,E1 -9409.821,E2 -9409.821} C_VEL
LIN {X 0,Y 432.311,Z 325.262,A -85,B 0,C 180,E1 -9413.022,E2 -9413.022} C_VEL
LIN {X 0,Y 432.363,Z 325.249,A -85,B 0,C 180,E1 -9415.996,E2 -9415.996} C_VEL
LIN {X 0,Y 432.351,Z 325.26,A -85,B 0,C 180,E1 -9419.489,E2 -9419.489} C_VEL
LIN {X 0,Y 432.386,Z 325.398,A -85,B 0,C 180,E1 -9420.414,E2 -9420.414} C_VEL
LIN {X 0,Y 435.928,Z 341.22,A -85,B 0,C 180,E1 -9423.423,E2 -9423.423} C_VEL
LIN {X 0,Y 436.407,Z 345.687,A -85,B 0,C 180,E1 -9424.226,E2 -9424.226} C_VEL
LIN {X 0,Y 435.114,Z 366.201,A -85,B 0,C 180,E1 -9427.692,E2 -9427.692} C_VEL
LIN {X 0,Y 435.041,Z 367.068,A -85,B 0,C 180,E1 -9427.837,E2 -9427.837} C_VEL
LIN {X 0,Y 439.743,Z 395.504,A -85,B 0,C 180,E1 -9428.551,E2 -9428.551} C_VEL
LIN {X 0,Y 438.284,Z 505.057,A -85,B 0,C 180,E1 -9430.382,E2 -9430.382} C_VEL
LIN {X 0,Y 437.754,Z 519.83,A -85,B 0,C 180,E1 -9430.814,E2 -9430.814} C_VEL
LIN {X 0,Y 437.162,Z 532.078,A -85,B 0,C 180,E1 -9431.329,E2 -9431.329} C_VEL
LIN {X 0,Y 436.385,Z 545.575,A -85,B 0,C 180,E1 -9432.086,E2 -9432.086} C_VEL
LIN {X 0,Y 435.492,Z 558.205,A -85,B 0,C 180,E1 -9432.991,E2 -9432.991} C_VEL
LIN {X 0,Y 434.659,Z 570.023,A -85,B 0,C 180,E1 -9434.045,E2 -9434.045} C_VEL
LIN {X 0,Y 433.805,Z 580.832,A -85,B 0,C 180,E1 -9435.216,E2 -9435.216} C_VEL
LIN {X 0,Y 433.076,Z 591.541,A -85,B 0,C 180,E1 -9436.629,E2 -9436.629} C_VEL
LIN {X 0,Y 432.447,Z 600.361,A -85,B 0,C 180,E1 -9438.04,E2 -9438.04} C_VEL
LIN {X 0,Y 431.956,Z 607.691,A -85,B 0,C 180,E1 -9439.452,E2 -9439.452} C_VEL
LIN {X 0,Y 431.589,Z 614.707,A -85,B 0,C 180,E1 -9441.1,E2 -9441.1} C_VEL
LIN {X 0,Y 431.392,Z 619.56,A -85,B 0,C 180,E1 -9442.51,E2 -9442.51} C_VEL
LIN {X 0,Y 431.263,Z 624.572,A -85,B 0,C 180,E1 -9444.388,E2 -9444.388} C_VEL
LIN {X 0,Y 431.182,Z 628.065,A -85,B 0,C 180,E1 -9446.261,E2 -9446.261} C_VEL
LIN {X 0,Y 431.264,Z 629.282,A -85,B 0,C 180,E1 -9447.197,E2 -9447.197} C_VEL
LIN {X 0,Y 431.191,Z 630.677,A -85,B 0,C 180,E1 -9449.065,E2 -9449.065} C_VEL
LIN {X 0,Y 431.191,Z 630.727,A -85,B 0,C 180,E1 -9450.933,E2 -9450.933} C_VEL
LIN {X 0,Y 431.233,Z 629.429,A -85,B 0,C 180,E1 -9452.802,E2 -9452.802} C_VEL
LIN {X 0,Y 431.244,Z 626.751,A -85,B 0,C 180,E1 -9454.673,E2 -9454.673} C_VEL
LIN {X 0,Y 431.372,Z 622.628,A -85,B 0,C 180,E1 -9456.548,E2 -9456.548} C_VEL
LIN {X 0,Y 431.517,Z 616.94,A -85,B 0,C 180,E1 -9458.428,E2 -9458.428} C_VEL
LIN {X 0,Y 431.86,Z 610.547,A -85,B 0,C 180,E1 -9460.074,E2 -9460.074} C_VEL
LIN {X 0,Y 432.466,Z 602.621,A -85,B 0,C 180,E1 -9461.72,E2 -9461.72} C_VEL
LIN {X 0,Y 433.007,Z 594.352,A -85,B 0,C 180,E1 -9463.133,E2 -9463.133} C_VEL
LIN {X 0,Y 433.774,Z 584.416,A -85,B 0,C 180,E1 -9464.543,E2 -9464.543} C_VEL
LIN {X 0,Y 434.695,Z 573.393,A -85,B 0,C 180,E1 -9465.832,E2 -9465.832} C_VEL
LIN {X 0,Y 435.743,Z 561.145,A -85,B 0,C 180,E1 -9466.997,E2 -9466.997} C_VEL
LIN {X 0,Y 436.657,Z 548.896,A -85,B 0,C 180,E1 -9467.936,E2 -9467.936} C_VEL
LIN {X 0,Y 437.493,Z 535.639,A -85,B 0,C 180,E1 -9468.74,E2 -9468.74} C_VEL
LIN {X 0,Y 438.295,Z 521.702,A -85,B 0,C 180,E1 -9469.372,E2 -9469.372} C_VEL
LIN {X 0,Y 438.926,Z 507.11,A -85,B 0,C 180,E1 -9469.83,E2 -9469.83} C_VEL
LIN {X 0,Y 439.374,Z 481.608,A -85,B 0,C 180,E1 -9470.297,E2 -9470.297} C_VEL
LIN {X 0,Y 440.535,Z 394.604,A -85,B 0,C 180,E1 -9471.763,E2 -9471.763} C_VEL
LIN {X 0,Y 436.556,Z 371.939,A -85,B 0,C 180,E1 -9472.397,E2 -9472.397} C_VEL
LIN {X 0,Y 435.483,Z 366.553,A -85,B 0,C 180,E1 -9472.568,E2 -9472.568} C_VEL
LIN {X 0,Y 436.822,Z 348.19,A -85,B 0,C 180,E1 -9475.746,E2 -9475.746} C_VEL
LIN {X 0,Y 436.893,Z 345.347,A -85,B 0,C 180,E1 -9476.254,E2 -9476.254} C_VEL
LIN {X 0,Y 434.525,Z 334.085,A -85,B 0,C 180,E1 -9478.483,E2 -9478.483} C_VEL
LIN {X 0,Y 432.345,Z 325.255,A -85,B 0,C 180,E1 -9480.338,E2 -9480.338} C_VEL
LIN {X 0,Y 432.357,Z 325.25,A -85,B 0,C 180,E1 -9484.003,E2 -9484.003} C_VEL
LIN {X 0,Y 432.33,Z 325.259,A -85,B 0,C 180,E1 -9487.198,E2 -9487.198} C_VEL
LIN {X 0,Y 432.352,Z 325.255,A -85,B 0,C 180,E1 -9490.182,E2 -9490.182} C_VEL
LIN {X 0,Y 432.313,Z 325.261,A -85,B 0,C 180,E1 -9493.06,E2 -9493.06} C_VEL
LIN {X 0,Y 432.335,Z 325.246,A -85,B 0,C 180,E1 -9495.663,E2 -9495.663} C_VEL
LIN {X 0,Y 432.357,Z 325.257,A -85,B 0,C 180,E1 -9498.393,E2 -9498.393} C_VEL
LIN {X 0,Y 432.339,Z 325.25,A -85,B 0,C 180,E1 -9501.85,E2 -9501.85} C_VEL
LIN {X 0,Y 432.335,Z 325.254,A -85,B 0,C 180,E1 -9505.322,E2 -9505.322} C_VEL
LIN {X 0,Y 432.32,Z 325.259,A -85,B 0,C 180,E1 -9508.654,E2 -9508.654} C_VEL
LIN {X 0,Y 432.374,Z 325.248,A -85,B 0,C 180,E1 -9511.368,E2 -9511.368} C_VEL
LIN {X 0,Y 432.356,Z 325.25,A -85,B 0,C 180,E1 -9513.967,E2 -9513.967} C_VEL
LIN {X 0,Y 432.311,Z 325.251,A -85,B 0,C 180,E1 -9517.035,E2 -9517.035} C_VEL
LIN {X 0,Y 432.379,Z 325.245,A -85,B 0,C 180,E1 -9520.514,E2 -9520.514} C_VEL
LIN {X 0,Y 432.435,Z 325.244,A -85,B 0,C 180,E1 -9523.961,E2 -9523.961} C_VEL
LIN {X 0,Y 432.45,Z 325.244,A -85,B 0,C 180,E1 -9527.803,E2 -9527.803} C_VEL
LIN {X 0,Y 432.483,Z 325.239,A -85,B 0,C 180,E1 -9531.59,E2 -9531.59} C_VEL
LIN {X 0,Y 432.582,Z 325.224,A -85,B 0,C 180,E1 -9534.406,E2 -9534.406} C_VEL
LIN {X 0,Y 432.587,Z 325.225,A -85,B 0,C 180,E1 -9538.138,E2 -9538.138} C_VEL
LIN {X 0,Y 432.61,Z 325.22,A -85,B 0,C 180,E1 -9540,E2 -9540} C_VEL
LIN {X 0,Y 432.57,Z 325.224,A -85,B 0,C 180,E1 -9542.793,E2 -9542.793} C_VEL
LIN {X 0,Y 432.497,Z 325.233,A -85,B 0,C 180,E1 -9546.531,E2 -9546.531} C_VEL
LIN {X 0,Y 432.414,Z 325.244,A -85,B 0,C 180,E1 -9549.353,E2 -9549.353} C_VEL
LIN {X 0,Y 432.42,Z 325.24,A -85,B 0,C 180,E1 -9552.803,E2 -9552.803} C_VEL
LIN {X 0,Y 432.384,Z 325.244,A -85,B 0,C 180,E1 -9556.47,E2 -9556.47} C_VEL
LIN {X 0,Y 432.327,Z 325.255,A -85,B 0,C 180,E1 -9559.961,E2 -9559.961} C_VEL
LIN {X 0,Y 432.306,Z 325.258,A -85,B 0,C 180,E1 -9562.965,E2 -9562.965} C_VEL
LIN {X 0,Y 432.327,Z 325.257,A -85,B 0,C 180,E1 -9565.002,E2 -9565.002} C_VEL
LIN {X 0,Y 432.329,Z 325.249,A -85,B 0,C 180,E1 -9568.127,E2 -9568.127} C_VEL
LIN {X 0,Y 432.31,Z 325.262,A -85,B 0,C 180,E1 -9571.346,E2 -9571.346} C_VEL
LIN {X 0,Y 432.328,Z 325.261,A -85,B 0,C 180,E1 -9574.678,E2 -9574.678} C_VEL
LIN {X 0,Y 432.326,Z 325.258,A -85,B 0,C 180,E1 -9578.151,E2 -9578.151} C_VEL
LIN {X 0,Y 432.324,Z 325.254,A -85,B 0,C 180,E1 -9581.602,E2 -9581.602} C_VEL
LIN {X 0,Y 432.325,Z 325.256,A -85,B 0,C 180,E1 -9584.348,E2 -9584.348} C_VEL
LIN {X 0,Y 432.366,Z 325.369,A -85,B 0,C 180,E1 -9586.541,E2 -9586.541} C_VEL
LIN {X 0,Y 435.034,Z 337.512,A -85,B 0,C 180,E1 -9589.401,E2 -9589.401} C_VEL
LIN {X 0,Y 435.149,Z 338.009,A -85,B 0,C 180,E1 -9589.477,E2 -9589.477} C_VEL
LIN {X 0,Y 437.955,Z 345.606,A -85,B 0,C 180,E1 -9589.787,E2 -9589.787} C_VEL
LIN {X 0,Y 440.992,Z 358.942,A -85,B 0,C 180,E1 -9590.205,E2 -9590.205} C_VEL
LIN {X 0,Y 439.309,Z 474.088,A -85,B 0,C 180,E1 -9592.164,E2 -9592.164} C_VEL
LIN {X 0,Y 438.795,Z 488.831,A -85,B 0,C 180,E1 -9592.608,E2 -9592.608} C_VEL
LIN {X 0,Y 438.2,Z 502.73,A -85,B 0,C 180,E1 -9593.226,E2 -9593.226} C_VEL
LIN {X 0,Y 437.465,Z 515.219,A -85,B 0,C 180,E1 -9593.958,E2 -9593.958} C_VEL
LIN {X 0,Y 436.577,Z 527.755,A -85,B 0,C 180,E1 -9594.89,E2 -9594.89} C_VEL
LIN {X 0,Y 435.596,Z 540.153,A -85,B 0,C 180,E1 -9596.039,E2 -9596.039} C_VEL
LIN {X 0,Y 434.79,Z 550.331,A -85,B 0,C 180,E1 -9597.196,E2 -9597.196} C_VEL
LIN {X 0,Y 433.946,Z 560.005,A -85,B 0,C 180,E1 -9598.514,E2 -9598.514} C_VEL
LIN {X 0,Y 433.144,Z 569.421,A -85,B 0,C 180,E1 -9600.072,E2 -9600.072} C_VEL
LIN {X 0,Y 432.523,Z 576.926,A -85,B 0,C 180,E1 -9601.593,E2 -9601.593} C_VEL
LIN {X 0,Y 432.015,Z 583.535,A -85,B 0,C 180,E1 -9603.247,E2 -9603.247} C_VEL
LIN {X 0,Y 431.655,Z 588.922,A -85,B 0,C 180,E1 -9604.957,E2 -9604.957} C_VEL
LIN {X 0,Y 431.434,Z 592.614,A -85,B 0,C 180,E1 -9606.479,E2 -9606.479} C_VEL
LIN {X 0,Y 431.242,Z 595.736,A -85,B 0,C 180,E1 -9608.268,E2 -9608.268} C_VEL
LIN {X 0,Y 431.124,Z 597.568,A -85,B 0,C 180,E1 -9610.031,E2 -9610.031} C_VEL
LIN {X 0,Y 430.429,Z 598.049,A -85,B 0,C 180,E1 -9610.809,E2 -9610.809} C_VEL
LIN {X 0,Y 427.548,Z 598.39,A -85,B 0,C 180,E1 -9612.077,E2 -9612.077} C_VEL
LIN {X 0,Y 425.137,Z 598.237,A -85,B 0,C 180,E1 -9613.099,E2 -9613.099} C_VEL
LIN {X 0,Y 424.115,Z 597.813,A -85,B 0,C 180,E1 -9613.886,E2 -9613.886} C_VEL
LIN {X 0,Y 424.038,Z 597.591,A -85,B 0,C 180,E1 -9614.152,E2 -9614.152} C_VEL
LIN {X 0,Y 424.085,Z 596.039,A -85,B 0,C 180,E1 -9615.607,E2 -9615.607} C_VEL
LIN {X 0,Y 424.328,Z 592.608,A -85,B 0,C 180,E1 -9617.567,E2 -9617.567} C_VEL
LIN {X 0,Y 424.581,Z 587.67,A -85,B 0,C 180,E1 -9619.51,E2 -9619.51} C_VEL
LIN {X 0,Y 424.897,Z 582.9,A -85,B 0,C 180,E1 -9620.96,E2 -9620.96} C_VEL
LIN {X 0,Y 425.4,Z 575.799,A -85,B 0,C 180,E1 -9622.686,E2 -9622.686} C_VEL
LIN {X 0,Y 426.067,Z 567.436,A -85,B 0,C 180,E1 -9624.321,E2 -9624.321} C_VEL
LIN {X 0,Y 426.728,Z 558.535,A -85,B 0,C 180,E1 -9625.751,E2 -9625.751} C_VEL
LIN {X 0,Y 427.448,Z 549.699,A -85,B 0,C 180,E1 -9626.938,E2 -9626.938} C_VEL
LIN {X 0,Y 428.276,Z 539.18,A -85,B 0,C 180,E1 -9628.12,E2 -9628.12} C_VEL
LIN {X 0,Y 429.134,Z 527.727,A -85,B 0,C 180,E1 -9629.18,E2 -9629.18} C_VEL
LIN {X 0,Y 429.97,Z 515.186,A -85,B 0,C 180,E1 -9630.118,E2 -9630.118} C_VEL
LIN {X 0,Y 430.743,Z 502.235,A -85,B 0,C 180,E1 -9630.877,E2 -9630.877} C_VEL
LIN {X 0,Y 431.294,Z 488.415,A -85,B 0,C 180,E1 -9631.489,E2 -9631.489} C_VEL
LIN {X 0,Y 431.761,Z 473.901,A -85,B 0,C 180,E1 -9631.925,E2 -9631.925} C_VEL
LIN {X 0,Y 433.31,Z 359.587,A -85,B 0,C 180,E1 -9633.869,E2 -9633.869} C_VEL
LIN {X 0,Y 429.422,Z 342.562,A -85,B 0,C 180,E1 -9634.359,E2 -9634.359} C_VEL
LIN {X 0,Y 427.641,Z 337.517,A -85,B 0,C 180,E1 -9634.552,E2 -9634.552} C_VEL
LIN {X 0,Y 425.471,Z 326.111,A -85,B 0,C 180,E1 -9637.115,E2 -9637.115} C_VEL
LIN {X 0,Y 425.359,Z 326.127,A -85,B 0,C 180,E1 -9640.472,E2 -9640.472} C_VEL
LIN {X 0,Y 425.362,Z 326.127,A -85,B 0,C 180,E1 -9643.375,E2 -9643.375} C_VEL
LIN {X 0,Y 425.359,Z 326.122,A -85,B 0,C 180,E1 -9646.605,E2 -9646.605} C_VEL
LIN {X 0,Y 425.327,Z 326.127,A -85,B 0,C 180,E1 -9649.636,E2 -9649.636} C_VEL
LIN {X 0,Y 425.286,Z 326.131,A -85,B 0,C 180,E1 -9652.34,E2 -9652.34} C_VEL
LIN {X 0,Y 425.257,Z 326.137,A -85,B 0,C 180,E1 -9655.449,E2 -9655.449} C_VEL
LIN {X 0,Y 425.298,Z 326.134,A -85,B 0,C 180,E1 -9658.859,E2 -9658.859} C_VEL
LIN {X 0,Y 425.245,Z 326.135,A -85,B 0,C 180,E1 -9661.929,E2 -9661.929} C_VEL
LIN {X 0,Y 425.289,Z 326.132,A -85,B 0,C 180,E1 -9665.338,E2 -9665.338} C_VEL
LIN {X 0,Y 425.274,Z 326.139,A -85,B 0,C 180,E1 -9668.902,E2 -9668.902} C_VEL
LIN {X 0,Y 425.254,Z 326.14,A -85,B 0,C 180,E1 -9672.656,E2 -9672.656} C_VEL
LIN {X 0,Y 425.283,Z 326.132,A -85,B 0,C 180,E1 -9675.284,E2 -9675.284} C_VEL
LIN {X 0,Y 425.245,Z 326.142,A -85,B 0,C 180,E1 -9678.618,E2 -9678.618} C_VEL
LIN {X 0,Y 425.268,Z 326.136,A -85,B 0,C 180,E1 -9682.305,E2 -9682.305} C_VEL
LIN {X 0,Y 425.285,Z 326.131,A -85,B 0,C 180,E1 -9685.816,E2 -9685.816} C_VEL
LIN {X 0,Y 425.289,Z 326.13,A -85,B 0,C 180,E1 -9689.24,E2 -9689.24} C_VEL
LIN {X 0,Y 425.248,Z 326.143,A -85,B 0,C 180,E1 -9692.436,E2 -9692.436} C_VEL
LIN {X 0,Y 425.322,Z 326.126,A -85,B 0,C 180,E1 -9695.601,E2 -9695.601} C_VEL
LIN {X 0,Y 425.29,Z 326.133,A -85,B 0,C 180,E1 -9698.682,E2 -9698.682} C_VEL
LIN {X 0,Y 425.314,Z 326.128,A -85,B 0,C 180,E1 -9701.702,E2 -9701.702} C_VEL
LIN {X 0,Y 425.305,Z 326.131,A -85,B 0,C 180,E1 -9704.669,E2 -9704.669} C_VEL
LIN {X 0,Y 425.414,Z 326.116,A -85,B 0,C 180,E1 -9707.599,E2 -9707.599} C_VEL
LIN {X 0,Y 425.41,Z 326.116,A -85,B 0,C 180,E1 -9711.45,E2 -9711.45} C_VEL
LIN {X 0,Y 425.536,Z 326.104,A -85,B 0,C 180,E1 -9714.313,E2 -9714.313} C_VEL
LIN {X 0,Y 425.574,Z 326.101,A -85,B 0,C 180,E1 -9718.108,E2 -9718.108} C_VEL
LIN {X 0,Y 425.698,Z 326.087,A -85,B 0,C 180,E1 -9720,E2 -9720} C_VEL
LIN {X 0,Y 425.535,Z 326.099,A -85,B 0,C 180,E1 -9722.84,E2 -9722.84} C_VEL
LIN {X 0,Y 425.543,Z 326.103,A -85,B 0,C 180,E1 -9725.687,E2 -9725.687} C_VEL
LIN {X 0,Y 425.44,Z 326.112,A -85,B 0,C 180,E1 -9728.55,E2 -9728.55} C_VEL
LIN {X 0,Y 425.416,Z 326.115,A -85,B 0,C 180,E1 -9732.402,E2 -9732.402} C_VEL
LIN {X 0,Y 425.392,Z 326.118,A -85,B 0,C 180,E1 -9736.312,E2 -9736.312} C_VEL
LIN {X 0,Y 425.333,Z 326.132,A -85,B 0,C 180,E1 -9739.636,E2 -9739.636} C_VEL
LIN {X 0,Y 425.309,Z 326.132,A -85,B 0,C 180,E1 -9743.365,E2 -9743.365} C_VEL
LIN {X 0,Y 425.351,Z 326.123,A -85,B 0,C 180,E1 -9746.844,E2 -9746.844} C_VEL
LIN {X 0,Y 425.295,Z 326.134,A -85,B 0,C 180,E1 -9749.72,E2 -9749.72} C_VEL
LIN {X 0,Y 425.286,Z 326.133,A -85,B 0,C 180,E1 -9753.048,E2 -9753.048} C_VEL
LIN {X 0,Y 425.285,Z 326.132,A -85,B 0,C 180,E1 -9755.928,E2 -9755.928} C_VEL
LIN {X 0,Y 425.301,Z 326.132,A -85,B 0,C 180,E1 -9759.043,E2 -9759.043} C_VEL
LIN {X 0,Y 425.282,Z 326.132,A -85,B 0,C 180,E1 -9762.652,E2 -9762.652} C_VEL
LIN {X 0,Y 425.265,Z 326.133,A -85,B 0,C 180,E1 -9766.044,E2 -9766.044} C_VEL
LIN {X 0,Y 425.278,Z 326.133,A -85,B 0,C 180,E1 -9768.621,E2 -9768.621} C_VEL
LIN {X 0,Y 425.31,Z 326.135,A -85,B 0,C 180,E1 -9771.102,E2 -9771.102} C_VEL
LIN {X 0,Y 425.303,Z 326.131,A -85,B 0,C 180,E1 -9774.664,E2 -9774.664} C_VEL
LIN {X 0,Y 425.269,Z 326.138,A -85,B 0,C 180,E1 -9778.073,E2 -9778.073} C_VEL
LIN {X 0,Y 425.324,Z 326.162,A -85,B 0,C 180,E1 -9780.112,E2 -9780.112} C_VEL
LIN {X 0,Y 428.925,Z 342.189,A -85,B 0,C 180,E1 -9783.218,E2 -9783.218} C_VEL
LIN {X 0,Y 429.502,Z 346.681,A -85,B 0,C 180,E1 -9784.045,E2 -9784.045} C_VEL
LIN {X 0,Y 428.223,Z 366.468,A -85,B 0,C 180,E1 -9787.441,E2 -9787.441} C_VEL
LIN {X 0,Y 428.178,Z 366.832,A -85,B 0,C 180,E1 -9787.502,E2 -9787.502} C_VEL
LIN {X 0,Y 433.063,Z 395.96,A -85,B 0,C 180,E1 -9788.248,E2 -9788.248} C_VEL
LIN {X 0,Y 431.544,Z 504.718,A -85,B 0,C 180,E1 -9790.094,E2 -9790.094} C_VEL
LIN {X 0,Y 430.988,Z 519.519,A -85,B 0,C 180,E1 -9790.532,E2 -9790.532} C_VEL
LIN {X 0,Y 430.351,Z 531.598,A -85,B 0,C 180,E1 -9791.044,E2 -9791.044} C_VEL
LIN {X 0,Y 429.595,Z 544.759,A -85,B 0,C 180,E1 -9791.788,E2 -9791.788} C_VEL
LIN {X 0,Y 428.668,Z 557.558,A -85,B 0,C 180,E1 -9792.712,E2 -9792.712} C_VEL
LIN {X 0,Y 427.727,Z 569.438,A -85,B 0,C 180,E1 -9793.779,E2 -9793.779} C_VEL
LIN {X 0,Y 426.844,Z 580.301,A -85,B 0,C 180,E1 -9794.969,E2 -9794.969} C_VEL
LIN {X 0,Y 426.09,Z 591.057,A -85,B 0,C 180,E1 -9796.405,E2 -9796.405} C_VEL
LIN {X 0,Y 425.446,Z 599.925,A -85,B 0,C 180,E1 -9797.841,E2 -9797.841} C_VEL
LIN {X 0,Y 424.931,Z 607.292,A -85,B 0,C 180,E1 -9799.276,E2 -9799.276} C_VEL
LIN {X 0,Y 424.533,Z 614.34,A -85,B 0,C 180,E1 -9800.951,E2 -9800.951} C_VEL
LIN {X 0,Y 424.321,Z 619.218,A -85,B 0,C 180,E1 -9802.385,E2 -9802.385} C_VEL
LIN {X 0,Y 424.174,Z 624.252,A -85,B 0,C 180,E1 -9804.294,E2 -9804.294} C_VEL
LIN {X 0,Y 424.168,Z 626.192,A -85,B 0,C 180,E1 -9805.247,E2 -9805.247} C_VEL
LIN {X 0,Y 424.16,Z 628.987,A -85,B 0,C 180,E1 -9807.15,E2 -9807.15} C_VEL
LIN {X 0,Y 424.109,Z 630.398,A -85,B 0,C 180,E1 -9809.05,E2 -9809.05} C_VEL
LIN {X 0,Y 424.109,Z 630.462,A -85,B 0,C 180,E1 -9810.949,E2 -9810.949} C_VEL
LIN {X 0,Y 424.13,Z 629.181,A -85,B 0,C 180,E1 -9812.849,E2 -9812.849} C_VEL
LIN {X 0,Y 424.17,Z 626.524,A -85,B 0,C 180,E1 -9814.751,E2 -9814.751} C_VEL
LIN {X 0,Y 424.294,Z 622.421,A -85,B 0,C 180,E1 -9816.657,E2 -9816.657} C_VEL
LIN {X 0,Y 424.453,Z 616.76,A -85,B 0,C 180,E1 -9818.569,E2 -9818.569} C_VEL
LIN {X 0,Y 424.805,Z 610.394,A -85,B 0,C 180,E1 -9820.244,E2 -9820.244} C_VEL
LIN {X 0,Y 425.463,Z 602.493,A -85,B 0,C 180,E1 -9821.915,E2 -9821.915} C_VEL
LIN {X 0,Y 426.174,Z 592.761,A -85,B 0,C 180,E1 -9823.59,E2 -9823.59} C_VEL
LIN {X 0,Y 427.014,Z 582.543,A -85,B 0,C 180,E1 -9825.023,E2 -9825.023} C_VEL
LIN {X 0,Y 428.091,Z 571.118,A -85,B 0,C 180,E1 -9826.327,E2 -9826.327} C_VEL
LIN {X 0,Y 429.08,Z 559.795,A -85,B 0,C 180,E1 -9827.392,E2 -9827.392} C_VEL
LIN {X 0,Y 430.02,Z 547.46,A -85,B 0,C 180,E1 -9828.336,E2 -9828.336} C_VEL
LIN {X 0,Y 430.933,Z 533.73,A -85,B 0,C 180,E1 -9829.159,E2 -9829.159} C_VEL
LIN {X 0,Y 431.774,Z 520.014,A -85,B 0,C 180,E1 -9829.77,E2 -9829.77} C_VEL
LIN {X 0,Y 432.378,Z 505.896,A -85,B 0,C 180,E1 -9830.205,E2 -9830.205} C_VEL
LIN {X 0,Y 433.035,Z 469.438,A -85,B 0,C 180,E1 -9830.856,E2 -9830.856} C_VEL
LIN {X 0,Y 434.006,Z 395.168,A -85,B 0,C 180,E1 -9832.132,E2 -9832.132} C_VEL
LIN {X 0,Y 429.659,Z 370.829,A -85,B 0,C 180,E1 -9832.839,E2 -9832.839} C_VEL
LIN {X 0,Y 428.759,Z 366.139,A -85,B 0,C 180,E1 -9833.011,E2 -9833.011} C_VEL
LIN {X 0,Y 430.134,Z 348.198,A -85,B 0,C 180,E1 -9836.176,E2 -9836.176} C_VEL
LIN {X 0,Y 428.743,Z 340.354,A -85,B 0,C 180,E1 -9837.727,E2 -9837.727} C_VEL
LIN {X 0,Y 425.336,Z 326.369,A -85,B 0,C 180,E1 -9840.67,E2 -9840.67} C_VEL
LIN {X 0,Y 425.285,Z 326.138,A -85,B 0,C 180,E1 -9840.815,E2 -9840.815} C_VEL
LIN {X 0,Y 425.309,Z 326.129,A -85,B 0,C 180,E1 -9844.287,E2 -9844.287} C_VEL
LIN {X 0,Y 425.285,Z 326.134,A -85,B 0,C 180,E1 -9847.692,E2 -9847.692} C_VEL
LIN {X 0,Y 425.296,Z 326.137,A -85,B 0,C 180,E1 -9850.522,E2 -9850.522} C_VEL
LIN {X 0,Y 425.253,Z 326.139,A -85,B 0,C 180,E1 -9853.35,E2 -9853.35} C_VEL
LIN {X 0,Y 425.259,Z 326.132,A -85,B 0,C 180,E1 -9856.647,E2 -9856.647} C_VEL
LIN {X 0,Y 425.281,Z 326.126,A -85,B 0,C 180,E1 -9859.872,E2 -9859.872} C_VEL
LIN {X 0,Y 425.279,Z 326.137,A -85,B 0,C 180,E1 -9862.486,E2 -9862.486} C_VEL
LIN {X 0,Y 425.302,Z 326.131,A -85,B 0,C 180,E1 -9865.816,E2 -9865.816} C_VEL
LIN {X 0,Y 425.296,Z 326.13,A -85,B 0,C 180,E1 -9869.235,E2 -9869.235} C_VEL
LIN {X 0,Y 425.344,Z 326.127,A -85,B 0,C 180,E1 -9872.442,E2 -9872.442} C_VEL
LIN {X 0,Y 425.342,Z 326.126,A -85,B 0,C 180,E1 -9875.601,E2 -9875.601} C_VEL
LIN {X 0,Y 425.285,Z 326.134,A -85,B 0,C 180,E1 -9878.681,E2 -9878.681} C_VEL
LIN {X 0,Y 425.325,Z 326.124,A -85,B 0,C 180,E1 -9881.702,E2 -9881.702} C_VEL
LIN {X 0,Y 425.348,Z 326.119,A -85,B 0,C 180,E1 -9884.67,E2 -9884.67} C_VEL
LIN {X 0,Y 425.403,Z 326.12,A -85,B 0,C 180,E1 -9887.598,E2 -9887.598} C_VEL
LIN {X 0,Y 425.433,Z 326.116,A -85,B 0,C 180,E1 -9891.449,E2 -9891.449} C_VEL
LIN {X 0,Y 425.539,Z 326.102,A -85,B 0,C 180,E1 -9894.313,E2 -9894.313} C_VEL
LIN {X 0,Y 425.556,Z 326.101,A -85,B 0,C 180,E1 -9898.107,E2 -9898.107} C_VEL
LIN {X 0,Y 425.562,Z 326.098,A -85,B 0,C 180,E1 -9900,E2 -9900} C_VEL
LIN {X 0,Y 425.523,Z 326.102,A -85,B 0,C 180,E1 -9902.84,E2 -9902.84} C_VEL
LIN {X 0,Y 425.459,Z 326.11,A -85,B 0,C 180,E1 -9906.64,E2 -9906.64} C_VEL
LIN {X 0,Y 425.375,Z 326.121,A -85,B 0,C 180,E1 -9909.51,E2 -9909.51} C_VEL
LIN {X 0,Y 425.383,Z 326.117,A -85,B 0,C 180,E1 -9912.903,E2 -9912.903} C_VEL
LIN {X 0,Y 425.336,Z 326.123,A -85,B 0,C 180,E1 -9916.598,E2 -9916.598} C_VEL
LIN {X 0,Y 425.318,Z 326.13,A -85,B 0,C 180,E1 -9919.635,E2 -9919.635} C_VEL
LIN {X 0,Y 425.293,Z 326.137,A -85,B 0,C 180,E1 -9923.365,E2 -9923.365} C_VEL
LIN {X 0,Y 425.287,Z 326.134,A -85,B 0,C 180,E1 -9926.499,E2 -9926.499} C_VEL
LIN {X 0,Y 425.273,Z 326.136,A -85,B 0,C 180,E1 -9929.72,E2 -9929.72} C_VEL
LIN {X 0,Y 425.272,Z 326.132,A -85,B 0,C 180,E1 -9933.048,E2 -9933.048} C_VEL
LIN {X 0,Y 425.272,Z 326.135,A -85,B 0,C 180,E1 -9935.929,E2 -9935.929} C_VEL
LIN {X 0,Y 425.272,Z 326.134,A -85,B 0,C 180,E1 -9939.041,E2 -9939.041} C_VEL
LIN {X 0,Y 425.281,Z 326.13,A -85,B 0,C 180,E1 -9941.959,E2 -9941.959} C_VEL
LIN {X 0,Y 425.276,Z 326.136,A -85,B 0,C 180,E1 -9945.284,E2 -9945.284} C_VEL
LIN {X 0,Y 425.316,Z 326.228,A -85,B 0,C 180,E1 -9946.163,E2 -9946.163} C_VEL
LIN {X 0,Y 427.942,Z 338.114,A -85,B 0,C 180,E1 -9949.017,E2 -9949.017} C_VEL
LIN {X 0,Y 431.814,Z 348.065,A -85,B 0,C 180,E1 -9949.451,E2 -9949.451} C_VEL
LIN {X 0,Y 434.527,Z 359.959,A -85,B 0,C 180,E1 -9949.837,E2 -9949.837} C_VEL
LIN {X 0,Y 432.752,Z 474.114,A -85,B 0,C 180,E1 -9951.807,E2 -9951.807} C_VEL
LIN {X 0,Y 432.241,Z 488.717,A -85,B 0,C 180,E1 -9952.248,E2 -9952.248} C_VEL
LIN {X 0,Y 431.652,Z 501.809,A -85,B 0,C 180,E1 -9952.827,E2 -9952.827} C_VEL
LIN {X 0,Y 430.842,Z 515.08,A -85,B 0,C 180,E1 -9953.606,E2 -9953.606} C_VEL
LIN {X 0,Y 429.966,Z 527.142,A -85,B 0,C 180,E1 -9954.507,E2 -9954.507} C_VEL
LIN {X 0,Y 428.974,Z 538.822,A -85,B 0,C 180,E1 -9955.584,E2 -9955.584} C_VEL
LIN {X 0,Y 427.985,Z 550.212,A -85,B 0,C 180,E1 -9956.874,E2 -9956.874} C_VEL
LIN {X 0,Y 427.081,Z 560.034,A -85,B 0,C 180,E1 -9958.226,E2 -9958.226} C_VEL
LIN {X 0,Y 426.227,Z 569.5,A -85,B 0,C 180,E1 -9959.809,E2 -9959.809} C_VEL
LIN {X 0,Y 425.549,Z 577.175,A -85,B 0,C 180,E1 -9961.385,E2 -9961.385} C_VEL
LIN {X 0,Y 425.046,Z 583.175,A -85,B 0,C 180,E1 -9962.895,E2 -9962.895} C_VEL
LIN {X 0,Y 424.65,Z 588.365,A -85,B 0,C 180,E1 -9964.514,E2 -9964.514} C_VEL
LIN {X 0,Y 424.413,Z 592.287,A -85,B 0,C 180,E1 -9966.085,E2 -9966.085} C_VEL
LIN {X 0,Y 424.167,Z 595.896,A -85,B 0,C 180,E1 -9968.102,E2 -9968.102} C_VEL
LIN {X 0,Y 424.032,Z 597.824,A -85,B 0,C 180,E1 -9970.021,E2 -9970.021} C_VEL
LIN {X 0,Y 424.019,Z 598.503,A -85,B 0,C 180,E1 -9971.645,E2 -9971.645} C_VEL
LIN {X 0,Y 424.02,Z 597.984,A -85,B 0,C 180,E1 -9973.635,E2 -9973.635} C_VEL
LIN {X 0,Y 424.038,Z 597.591,A -85,B 0,C 180,E1 -9974.152,E2 -9974.152} C_VEL
LIN {X 0,Y 423.398,Z 596.875,A -85,B 0,C 180,E1 -9974.939,E2 -9974.939} C_VEL
LIN {X 0,Y 420.611,Z 595.285,A -85,B 0,C 180,E1 -9976.211,E2 -9976.211} C_VEL
LIN {X 0,Y 418.29,Z 593.628,A -85,B 0,C 180,E1 -9977.227,E2 -9977.227} C_VEL
LIN {X 0,Y 417.356,Z 592.054,A -85,B 0,C 180,E1 -9978.003,E2 -9978.003} C_VEL
LIN {X 0,Y 417.313,Z 591.479,A -85,B 0,C 180,E1 -9978.264,E2 -9978.264} C_VEL
LIN {X 0,Y 417.567,Z 587.302,A -85,B 0,C 180,E1 -9979.822,E2 -9979.822} C_VEL
LIN {X 0,Y 417.934,Z 582.359,A -85,B 0,C 180,E1 -9981.296,E2 -9981.296} C_VEL
LIN {X 0,Y 418.426,Z 575.473,A -85,B 0,C 180,E1 -9982.963,E2 -9982.963} C_VEL
LIN {X 0,Y 419.06,Z 567.865,A -85,B 0,C 180,E1 -9984.467,E2 -9984.467} C_VEL
LIN {X 0,Y 419.778,Z 558.989,A -85,B 0,C 180,E1 -9985.921,E2 -9985.921} C_VEL
LIN {X 0,Y 420.508,Z 550.193,A -85,B 0,C 180,E1 -9987.127,E2 -9987.127} C_VEL
LIN {X 0,Y 421.371,Z 539.705,A -85,B 0,C 180,E1 -9988.329,E2 -9988.329} C_VEL
LIN {X 0,Y 422.27,Z 528.054,A -85,B 0,C 180,E1 -9989.425,E2 -9989.425} C_VEL
LIN {X 0,Y 423.139,Z 515.803,A -85,B 0,C 180,E1 -9990.358,E2 -9990.358} C_VEL
LIN {X 0,Y 423.935,Z 502.937,A -85,B 0,C 180,E1 -9991.129,E2 -9991.129} C_VEL
LIN {X 0,Y 424.534,Z 489.225,A -85,B 0,C 180,E1 -9991.75,E2 -9991.75} C_VEL
LIN {X 0,Y 424.966,Z 475.049,A -85,B 0,C 180,E1 -9992.193,E2 -9992.193} C_VEL
LIN {X 0,Y 426.018,Z 405.343,A -85,B 0,C 180,E1 -9993.41,E2 -9993.41} C_VEL
LIN {X 0,Y 426.533,Z 359.902,A -85,B 0,C 180,E1 -9994.194,E2 -9994.194} C_VEL
LIN {X 0,Y 423.06,Z 345.039,A -85,B 0,C 180,E1 -9994.635,E2 -9994.635} C_VEL
LIN {X 0,Y 420.521,Z 337.735,A -85,B 0,C 180,E1 -9994.914,E2 -9994.914} C_VEL
LIN {X 0,Y 418.431,Z 326.989,A -85,B 0,C 180,E1 -9997.414,E2 -9997.414} C_VEL
LIN {X 0,Y 418.328,Z 327.004,A -85,B 0,C 180,E1 -10000.65,E2 -10000.65} C_VEL
LIN {X 0,Y 418.31,Z 327.003,A -85,B 0,C 180,E1 -10003.605,E2 -10003.605} C_VEL
LIN {X 0,Y 418.311,Z 327.001,A -85,B 0,C 180,E1 -10006.736,E2 -10006.736} C_VEL
LIN {X 0,Y 418.269,Z 327.005,A -85,B 0,C 180,E1 -10009.791,E2 -10009.791} C_VEL
LIN {X 0,Y 418.226,Z 327.013,A -85,B 0,C 180,E1 -10012.738,E2 -10012.738} C_VEL
LIN {X 0,Y 418.216,Z 327.011,A -85,B 0,C 180,E1 -10015.908,E2 -10015.908} C_VEL
LIN {X 0,Y 418.255,Z 327.012,A -85,B 0,C 180,E1 -10019.163,E2 -10019.163} C_VEL
LIN {X 0,Y 418.229,Z 327.012,A -85,B 0,C 180,E1 -10022.53,E2 -10022.53} C_VEL
LIN {X 0,Y 418.247,Z 327.014,A -85,B 0,C 180,E1 -10024.843,E2 -10024.843} C_VEL
LIN {X 0,Y 418.232,Z 327.012,A -85,B 0,C 180,E1 -10028.445,E2 -10028.445} C_VEL
LIN {X 0,Y 418.217,Z 327.012,A -85,B 0,C 180,E1 -10032.237,E2 -10032.237} C_VEL
LIN {X 0,Y 418.234,Z 327.012,A -85,B 0,C 180,E1 -10035.109,E2 -10035.109} C_VEL
LIN {X 0,Y 418.217,Z 327.011,A -85,B 0,C 180,E1 -10037.764,E2 -10037.764} C_VEL
LIN {X 0,Y 418.227,Z 327.01,A -85,B 0,C 180,E1 -10041.556,E2 -10041.556} C_VEL
LIN {X 0,Y 418.249,Z 327.008,A -85,B 0,C 180,E1 -10045.159,E2 -10045.159} C_VEL
LIN {X 0,Y 418.244,Z 327.008,A -85,B 0,C 180,E1 -10047.472,E2 -10047.472} C_VEL
LIN {X 0,Y 418.26,Z 327.008,A -85,B 0,C 180,E1 -10050.899,E2 -10050.899} C_VEL
LIN {X 0,Y 418.219,Z 327.014,A -85,B 0,C 180,E1 -10054.093,E2 -10054.093} C_VEL
LIN {X 0,Y 418.227,Z 327.01,A -85,B 0,C 180,E1 -10057.264,E2 -10057.264} C_VEL
LIN {X 0,Y 418.284,Z 327.01,A -85,B 0,C 180,E1 -10060.365,E2 -10060.365} C_VEL
LIN {X 0,Y 418.281,Z 327.003,A -85,B 0,C 180,E1 -10063.404,E2 -10063.404} C_VEL
LIN {X 0,Y 418.349,Z 326.995,A -85,B 0,C 180,E1 -10067,E2 -10067} C_VEL
LIN {X 0,Y 418.34,Z 327.001,A -85,B 0,C 180,E1 -10070.329,E2 -10070.329} C_VEL
LIN {X 0,Y 418.448,Z 326.982,A -85,B 0,C 180,E1 -10073.249,E2 -10073.249} C_VEL
LIN {X 0,Y 418.332,Z 326.997,A -85,B 0,C 180,E1 -10075.182,E2 -10075.182} C_VEL
LIN {X 0,Y 418.543,Z 326.977,A -85,B 0,C 180,E1 -10078.076,E2 -10078.076} C_VEL
LIN {X 0,Y 418.667,Z 326.962,A -85,B 0,C 180,E1 -10080,E2 -10080} C_VEL
LIN {X 0,Y 418.491,Z 326.977,A -85,B 0,C 180,E1 -10082.888,E2 -10082.888} C_VEL
LIN {X 0,Y 418.501,Z 326.982,A -85,B 0,C 180,E1 -10085.783,E2 -10085.783} C_VEL
LIN {X 0,Y 418.4,Z 326.988,A -85,B 0,C 180,E1 -10088.695,E2 -10088.695} C_VEL
LIN {X 0,Y 418.318,Z 327.004,A -85,B 0,C 180,E1 -10091.631,E2 -10091.631} C_VEL
LIN {X 0,Y 418.306,Z 327,A -85,B 0,C 180,E1 -10094.597,E2 -10094.597} C_VEL
LIN {X 0,Y 418.292,Z 327.008,A -85,B 0,C 180,E1 -10097.604,E2 -10097.604} C_VEL
LIN {X 0,Y 418.254,Z 327.006,A -85,B 0,C 180,E1 -10100.663,E2 -10100.663} C_VEL
LIN {X 0,Y 418.289,Z 327.007,A -85,B 0,C 180,E1 -10103.781,E2 -10103.781} C_VEL
LIN {X 0,Y 418.315,Z 327.001,A -85,B 0,C 180,E1 -10107.07,E2 -10107.07} C_VEL
LIN {X 0,Y 418.249,Z 327.007,A -85,B 0,C 180,E1 -10110.272,E2 -10110.272} C_VEL
LIN {X 0,Y 418.252,Z 327.011,A -85,B 0,C 180,E1 -10113.677,E2 -10113.677} C_VEL
LIN {X 0,Y 418.243,Z 327.013,A -85,B 0,C 180,E1 -10117.224,E2 -10117.224} C_VEL
LIN {X 0,Y 418.255,Z 327.009,A -85,B 0,C 180,E1 -10119.682,E2 -10119.682} C_VEL
LIN {X 0,Y 418.236,Z 327.009,A -85,B 0,C 180,E1 -10122.321,E2 -10122.321} C_VEL
LIN {X 0,Y 418.242,Z 327.014,A -85,B 0,C 180,E1 -10125.109,E2 -10125.109} C_VEL
LIN {X 0,Y 418.244,Z 327.009,A -85,B 0,C 180,E1 -10127.767,E2 -10127.767} C_VEL
LIN {X 0,Y 418.257,Z 327.008,A -85,B 0,C 180,E1 -10130.619,E2 -10130.619} C_VEL
LIN {X 0,Y 418.247,Z 327.007,A -85,B 0,C 180,E1 -10133.975,E2 -10133.975} C_VEL
LIN {X 0,Y 418.262,Z 327.012,A -85,B 0,C 180,E1 -10137.156,E2 -10137.156} C_VEL
LIN {X 0,Y 418.292,Z 327.052,A -85,B 0,C 180,E1 -10139.828,E2 -10139.828} C_VEL
LIN {X 0,Y 422.195,Z 344.641,A -85,B 0,C 180,E1 -10143.291,E2 -10143.291} C_VEL
LIN {X 0,Y 422.565,Z 348.738,A -85,B 0,C 180,E1 -10144.047,E2 -10144.047} C_VEL
LIN {X 0,Y 421.328,Z 366.555,A -85,B 0,C 180,E1 -10147.156,E2 -10147.156} C_VEL
LIN {X 0,Y 426.273,Z 396.154,A -85,B 0,C 180,E1 -10147.931,E2 -10147.931} C_VEL
LIN {X 0,Y 424.776,Z 504.24,A -85,B 0,C 180,E1 -10149.794,E2 -10149.794} C_VEL
LIN {X 0,Y 424.241,Z 518.379,A -85,B 0,C 180,E1 -10150.21,E2 -10150.21} C_VEL
LIN {X 0,Y 423.529,Z 531.727,A -85,B 0,C 180,E1 -10150.783,E2 -10150.783} C_VEL
LIN {X 0,Y 422.702,Z 545.487,A -85,B 0,C 180,E1 -10151.584,E2 -10151.584} C_VEL
LIN {X 0,Y 421.71,Z 558.347,A -85,B 0,C 180,E1 -10152.543,E2 -10152.543} C_VEL
LIN {X 0,Y 420.763,Z 570.043,A -85,B 0,C 180,E1 -10153.628,E2 -10153.628} C_VEL
LIN {X 0,Y 419.778,Z 581.746,A -85,B 0,C 180,E1 -10154.959,E2 -10154.959} C_VEL
LIN {X 0,Y 418.999,Z 592.213,A -85,B 0,C 180,E1 -10156.418,E2 -10156.418} C_VEL
LIN {X 0,Y 418.337,Z 600.842,A -85,B 0,C 180,E1 -10157.877,E2 -10157.877} C_VEL
LIN {X 0,Y 417.74,Z 609.077,A -85,B 0,C 180,E1 -10159.58,E2 -10159.58} C_VEL
LIN {X 0,Y 417.393,Z 615.71,A -85,B 0,C 180,E1 -10161.283,E2 -10161.283} C_VEL
LIN {X 0,Y 417.155,Z 621.586,A -85,B 0,C 180,E1 -10163.226,E2 -10163.226} C_VEL
LIN {X 0,Y 417.073,Z 625.866,A -85,B 0,C 180,E1 -10165.166,E2 -10165.166} C_VEL
LIN {X 0,Y 417.057,Z 628.683,A -85,B 0,C 180,E1 -10167.101,E2 -10167.101} C_VEL
LIN {X 0,Y 417.03,Z 630.115,A -85,B 0,C 180,E1 -10169.034,E2 -10169.034} C_VEL
LIN {X 0,Y 417.03,Z 630.198,A -85,B 0,C 180,E1 -10170.965,E2 -10170.965} C_VEL
LIN {X 0,Y 417.027,Z 628.938,A -85,B 0,C 180,E1 -10172.897,E2 -10172.897} C_VEL
LIN {X 0,Y 417.076,Z 626.306,A -85,B 0,C 180,E1 -10174.832,E2 -10174.832} C_VEL
LIN {X 0,Y 417.226,Z 622.224,A -85,B 0,C 180,E1 -10176.771,E2 -10176.771} C_VEL
LIN {X 0,Y 417.403,Z 616.584,A -85,B 0,C 180,E1 -10178.715,E2 -10178.715} C_VEL
LIN {X 0,Y 417.774,Z 610.24,A -85,B 0,C 180,E1 -10180.418,E2 -10180.418} C_VEL
LIN {X 0,Y 418.461,Z 602.365,A -85,B 0,C 180,E1 -10182.118,E2 -10182.118} C_VEL
LIN {X 0,Y 419.107,Z 594.168,A -85,B 0,C 180,E1 -10183.577,E2 -10183.577} C_VEL
LIN {X 0,Y 419.957,Z 584.321,A -85,B 0,C 180,E1 -10185.033,E2 -10185.033} C_VEL
LIN {X 0,Y 421.03,Z 573.408,A -85,B 0,C 180,E1 -10186.36,E2 -10186.36} C_VEL
LIN {X 0,Y 422.192,Z 561.331,A -85,B 0,C 180,E1 -10187.56,E2 -10187.56} C_VEL
LIN {X 0,Y 423.17,Z 549.583,A -85,B 0,C 180,E1 -10188.507,E2 -10188.507} C_VEL
LIN {X 0,Y 424.099,Z 536.38,A -85,B 0,C 180,E1 -10189.355,E2 -10189.355} C_VEL
LIN {X 0,Y 424.972,Z 522.925,A -85,B 0,C 180,E1 -10190.005,E2 -10190.005} C_VEL
LIN {X 0,Y 425.714,Z 509.236,A -85,B 0,C 180,E1 -10190.473,E2 -10190.473} C_VEL
LIN {X 0,Y 426.095,Z 492.319,A -85,B 0,C 180,E1 -10190.832,E2 -10190.832} C_VEL
LIN {X 0,Y 427.601,Z 396.627,A -85,B 0,C 180,E1 -10192.49,E2 -10192.49} C_VEL
LIN {X 0,Y 423.379,Z 372.736,A -85,B 0,C 180,E1 -10193.202,E2 -10193.202} C_VEL
LIN {X 0,Y 422.024,Z 365.91,A -85,B 0,C 180,E1 -10193.437,E2 -10193.437} C_VEL
LIN {X 0,Y 423.277,Z 350.074,A -85,B 0,C 180,E1 -10196.284,E2 -10196.284} C_VEL
LIN {X 0,Y 422.016,Z 342.57,A -85,B 0,C 180,E1 -10197.793,E2 -10197.793} C_VEL
LIN {X 0,Y 418.723,Z 328.902,A -85,B 0,C 180,E1 -10200.719,E2 -10200.719} C_VEL
LIN {X 0,Y 418.219,Z 327.018,A -85,B 0,C 180,E1 -10201.162,E2 -10201.162} C_VEL
LIN {X 0,Y 418.246,Z 327.008,A -85,B 0,C 180,E1 -10203.676,E2 -10203.676} C_VEL
LIN {X 0,Y 418.244,Z 327.014,A -85,B 0,C 180,E1 -10207.222,E2 -10207.222} C_VEL
LIN {X 0,Y 418.261,Z 327.009,A -85,B 0,C 180,E1 -10209.679,E2 -10209.679} C_VEL
LIN {X 0,Y 418.241,Z 327.005,A -85,B 0,C 180,E1 -10212.322,E2 -10212.322} C_VEL
LIN {X 0,Y 418.234,Z 327.005,A -85,B 0,C 180,E1 -10215.108,E2 -10215.108} C_VEL
LIN {X 0,Y 418.238,Z 327.011,A -85,B 0,C 180,E1 -10217.766,E2 -10217.766} C_VEL
LIN {X 0,Y 418.249,Z 327,A -85,B 0,C 180,E1 -10220.618,E2 -10220.618} C_VEL
LIN {X 0,Y 418.24,Z 327.011,A -85,B 0,C 180,E1 -10223.975,E2 -10223.975} C_VEL
LIN {X 0,Y 418.251,Z 327.005,A -85,B 0,C 180,E1 -10227.155,E2 -10227.155} C_VEL
LIN {X 0,Y 418.268,Z 327.007,A -85,B 0,C 180,E1 -10230.838,E2 -10230.838} C_VEL
LIN {X 0,Y 418.263,Z 327.006,A -85,B 0,C 180,E1 -10234.095,E2 -10234.095} C_VEL
LIN {X 0,Y 418.224,Z 327.006,A -85,B 0,C 180,E1 -10237.263,E2 -10237.263} C_VEL
LIN {X 0,Y 418.276,Z 327.003,A -85,B 0,C 180,E1 -10240.364,E2 -10240.364} C_VEL
LIN {X 0,Y 418.318,Z 327.001,A -85,B 0,C 180,E1 -10243.404,E2 -10243.404} C_VEL
LIN {X 0,Y 418.338,Z 326.998,A -85,B 0,C 180,E1 -10246.999,E2 -10246.999} C_VEL
LIN {X 0,Y 418.33,Z 327.001,A -85,B 0,C 180,E1 -10250.328,E2 -10250.328} C_VEL
LIN {X 0,Y 418.505,Z 326.974,A -85,B 0,C 180,E1 -10252.279,E2 -10252.279} C_VEL
LIN {X 0,Y 418.499,Z 326.98,A -85,B 0,C 180,E1 -10254.217,E2 -10254.217} C_VEL
LIN {X 0,Y 418.525,Z 326.977,A -85,B 0,C 180,E1 -10258.075,E2 -10258.075} C_VEL
LIN {X 0,Y 418.397,Z 326.987,A -85,B 0,C 180,E1 -10260.962,E2 -10260.962} C_VEL
LIN {X 0,Y 418.479,Z 326.98,A -85,B 0,C 180,E1 -10262.888,E2 -10262.888} C_VEL
LIN {X 0,Y 418.425,Z 326.986,A -85,B 0,C 180,E1 -10266.752,E2 -10266.752} C_VEL
LIN {X 0,Y 418.316,Z 327.001,A -85,B 0,C 180,E1 -10269.672,E2 -10269.672} C_VEL
LIN {X 0,Y 418.336,Z 326.995,A -85,B 0,C 180,E1 -10273,E2 -10273} C_VEL
LIN {X 0,Y 418.295,Z 327,A -85,B 0,C 180,E1 -10276.732,E2 -10276.732} C_VEL
LIN {X 0,Y 418.26,Z 327.009,A -85,B 0,C 180,E1 -10279.79,E2 -10279.79} C_VEL
LIN {X 0,Y 418.227,Z 327.009,A -85,B 0,C 180,E1 -10282.736,E2 -10282.736} C_VEL
LIN {X 0,Y 418.225,Z 327.014,A -85,B 0,C 180,E1 -10285.907,E2 -10285.907} C_VEL
LIN {X 0,Y 418.249,Z 327.003,A -85,B 0,C 180,E1 -10289.163,E2 -10289.163} C_VEL
LIN {X 0,Y 418.247,Z 327.007,A -85,B 0,C 180,E1 -10292.844,E2 -10292.844} C_VEL
LIN {X 0,Y 418.235,Z 327.011,A -85,B 0,C 180,E1 -10296.238,E2 -10296.238} C_VEL
LIN {X 0,Y 418.235,Z 327.008,A -85,B 0,C 180,E1 -10299.683,E2 -10299.683} C_VEL
LIN {X 0,Y 418.22,Z 327.011,A -85,B 0,C 180,E1 -10302.322,E2 -10302.322} C_VEL
LIN {X 0,Y 418.269,Z 327.196,A -85,B 0,C 180,E1 -10305.795,E2 -10305.795} C_VEL
LIN {X 0,Y 420.875,Z 338.619,A -85,B 0,C 180,E1 -10308.562,E2 -10308.562} C_VEL
LIN {X 0,Y 425.618,Z 350.309,A -85,B 0,C 180,E1 -10309.096,E2 -10309.096} C_VEL
LIN {X 0,Y 428.114,Z 361.362,A -85,B 0,C 180,E1 -10309.463,E2 -10309.463} C_VEL
LIN {X 0,Y 426.19,Z 475.168,A -85,B 0,C 180,E1 -10311.464,E2 -10311.464} C_VEL
LIN {X 0,Y 425.673,Z 489.161,A -85,B 0,C 180,E1 -10311.899,E2 -10311.899} C_VEL
LIN {X 0,Y 424.989,Z 503.204,A -85,B 0,C 180,E1 -10312.539,E2 -10312.539} C_VEL
LIN {X 0,Y 424.084,Z 516.908,A -85,B 0,C 180,E1 -10313.375,E2 -10313.375} C_VEL
LIN {X 0,Y 423.136,Z 528.939,A -85,B 0,C 180,E1 -10314.311,E2 -10314.311} C_VEL
LIN {X 0,Y 422.126,Z 540.114,A -85,B 0,C 180,E1 -10315.38,E2 -10315.38} C_VEL
LIN {X 0,Y 421.092,Z 551.597,A -85,B 0,C 180,E1 -10316.725,E2 -10316.725} C_VEL
LIN {X 0,Y 420.092,Z 561.863,A -85,B 0,C 180,E1 -10318.199,E2 -10318.199} C_VEL
